C03628=1010.077,358.857,339.803,170.811,52.847,160.488
C03629=1010.084,359.105,339.765,170.821,52.843,160.489
C03630=1010.090,359.351,339.728,170.830,52.838,160.489
C03631=1010.098,359.598,339.690,170.839,52.835,160.490
C03632=1010.105,359.846,339.653,170.848,52.830,160.491
C03633=1010.112,360.093,339.616,170.857,52.827,160.492
C03634=1010.119,360.340,339.578,170.866,52.823,160.493
C03635=1010.126,360.587,339.541,170.876,52.819,160.494
C03636=1010.133,360.834,339.504,170.884,52.814,160.495
C03637=1010.140,361.081,339.466,170.893,52.811,160.495
C03638=1010.147,361.328,339.429,170.903,52.806,160.496
C03639=1010.155,361.575,339.391,170.912,52.803,160.497
C03640=1010.162,361.822,339.354,170.922,52.799,160.498
C03641=1010.169,362.069,339.316,170.930,52.795,160.499
C03642=1010.176,362.317,339.279,170.939,52.791,160.500
C03643=1010.184,362.564,339.241,170.949,52.787,160.501
C03644=1010.191,362.811,339.204,170.958,52.783,160.502
C03645=1010.198,363.058,339.166,170.968,52.779,160.503
C03646=1010.205,363.305,339.128,170.977,52.775,160.504
C03647=1010.213,363.552,339.090,170.987,52.771,160.505
C03648=1010.220,363.799,339.053,170.995,52.767,160.505
C03649=1010.227,364.046,339.015,171.005,52.763,160.506
C03650=1010.235,364.293,338.978,171.014,52.760,160.507
C03651=1010.242,364.539,338.939,171.023,52.756,160.508
C03652=1010.250,364.787,338.902,171.033,52.752,160.509
C03653=1010.257,365.034,338.864,171.042,52.749,160.510
C03654=1010.265,365.281,338.826,171.052,52.745,160.511
C03655=1010.272,365.528,338.788,171.061,52.741,160.512
C03656=1009.942,363.417,338.757,170.962,52.829,160.514
C03657=1009.935,363.169,338.794,170.952,52.833,160.513
C03658=1009.928,362.922,338.832,170.943,52.836,160.512
C03659=1009.920,362.675,338.869,170.934,52.840,160.511
C03660=1009.913,362.428,338.907,170.924,52.844,160.510
C03661=1009.906,362.181,338.944,170.915,52.848,160.509
C03662=1009.899,361.934,338.982,170.905,52.852,160.508
C03663=1009.891,361.687,339.019,170.897,52.856,160.508
C03664=1009.884,361.439,339.057,170.887,52.860,160.507
C03665=1009.877,361.192,339.094,170.878,52.864,160.506
C03666=1009.870,360.945,339.132,170.869,52.868,160.505
C03667=1009.863,360.698,339.169,170.859,52.872,160.504
C03668=1009.856,360.452,339.207,170.851,52.876,160.503
C03669=1009.849,360.205,339.244,170.842,52.880,160.502
C03670=1009.841,359.957,339.282,170.832,52.884,160.501
C03671=1009.834,359.710,339.318,170.823,52.888,160.501
C03672=1009.827,359.462,339.356,170.814,52.892,160.500
C03673=1009.821,359.216,339.393,170.805,52.896,160.499
C03674=1009.813,358.969,339.431,170.796,52.900,160.498
C03675=1009.806,358.721,339.468,170.786,52.904,160.497
C03676=1009.800,358.475,339.505,170.778,52.908,160.496
C03677=1009.793,358.227,339.541,170.769,52.913,160.496
C03678=1009.786,357.980,339.579,170.759,52.917,160.495
C03679=1009.779,357.733,339.615,170.751,52.921,160.494
C03680=1009.772,357.486,339.653,170.742,52.925,160.493
C03681=1009.765,357.238,339.690,170.733,52.929,160.492
C03682=1009.758,356.992,339.726,170.723,52.933,160.491
C03683=1009.751,356.744,339.763,170.715,52.937,160.491
C03684=1009.744,356.496,339.800,170.706,52.942,160.490
C03685=1009.737,356.250,339.837,170.697,52.946,160.489
C03686=1009.729,356.002,339.873,170.688,52.950,160.488
C03687=1009.723,355.755,339.910,170.679,52.954,160.487
C03688=1009.716,355.508,339.947,170.670,52.959,160.487
C03689=1009.710,355.284,339.979,170.662,52.962,160.486
C03690=1009.704,355.060,340.012,170.655,52.966,160.485
C03691=1009.697,354.837,340.046,170.646,52.970,160.485
C03692=1009.691,354.612,340.079,170.639,52.974,160.484
C03693=1009.684,354.389,340.112,170.630,52.978,160.483
C03694=1009.678,354.165,340.145,170.623,52.982,160.483
C03695=1009.673,353.941,340.178,170.615,52.986,160.482
C03696=1009.666,353.717,340.211,170.606,52.990,160.481
C03697=1009.660,353.470,340.247,170.598,52.994,160.481
C03698=1009.653,353.223,340.284,170.589,52.999,160.480
C03699=1009.646,352.976,340.320,170.581,53.003,160.479
C03700=1009.639,352.728,340.356,170.571,53.008,160.478
C03701=1009.633,352.480,340.392,170.563,53.012,160.478
C03702=1009.625,352.234,340.428,170.554,53.016,160.477
C03703=1009.619,351.986,340.465,170.546,53.020,160.476
C03704=1009.611,351.739,340.501,170.537,53.025,160.476
C03705=1009.605,351.492,340.536,170.528,53.030,160.475
C03706=1009.598,351.244,340.573,170.519,53.034,160.474
C03707=1009.591,350.997,340.609,170.511,53.038,160.474
C03708=1009.585,350.750,340.644,170.503,53.043,160.473
C03709=1009.578,350.503,340.681,170.494,53.047,160.472
C03710=1009.571,350.255,340.716,170.485,53.052,160.472
C03711=1009.565,350.008,340.753,170.477,53.057,160.471
C03712=1009.558,349.760,340.788,170.468,53.061,160.470
C03713=1009.552,349.513,340.824,170.459,53.065,160.470
C03714=1009.545,349.266,340.859,170.451,53.070,160.469
C03715=1009.538,349.019,340.896,170.443,53.074,160.468
C03716=1009.531,348.771,340.931,170.434,53.079,160.468
C03717=1009.525,348.524,340.968,170.425,53.084,160.467
C03718=1009.518,348.276,341.003,170.417,53.089,160.467
C03719=1009.512,348.029,341.039,170.409,53.093,160.466
C03720=1009.505,347.782,341.074,170.400,53.098,160.465
C03721=1009.499,347.534,341.110,170.392,53.102,160.465
C03722=1009.492,347.287,341.145,170.384,53.107,160.464
C03723=1009.486,347.039,341.181,170.374,53.111,160.463
C03724=1009.479,346.792,341.217,170.366,53.116,160.463
C03725=1009.472,346.545,341.252,170.358,53.121,160.462
C03726=1009.466,346.297,341.288,170.349,53.125,160.462
C03727=1009.459,346.050,341.323,170.341,53.130,160.461
C03728=1009.453,345.802,341.359,170.333,53.135,160.461
C03729=1009.447,345.555,341.394,170.325,53.139,160.460
C03730=1009.440,345.308,341.429,170.317,53.144,160.459
C03731=1009.434,345.060,341.465,170.309,53.149,160.459
C03732=1009.427,344.812,341.500,170.300,53.154,160.458
C03733=1009.420,344.565,341.535,170.291,53.159,160.457
C03734=1009.413,344.318,341.570,170.283,53.163,160.457
C03735=1009.408,344.071,341.605,170.275,53.168,160.456
C03736=1009.402,343.823,341.640,170.267,53.173,160.456
C03737=1009.395,343.575,341.675,170.259,53.178,160.455
C03738=1009.388,343.328,341.710,170.250,53.183,160.455
C03739=1009.381,343.081,341.745,170.242,53.187,160.454
C03740=1009.376,342.832,341.780,170.234,53.192,160.454
C03741=1009.369,342.586,341.815,170.226,53.197,160.453
C03742=1009.363,342.338,341.850,170.218,53.202,160.453
C03743=1009.356,342.090,341.885,170.209,53.207,160.452
C03744=1009.350,341.843,341.920,170.201,53.212,160.452
C03745=1009.344,341.596,341.955,170.193,53.216,160.451
C03746=1009.337,341.348,341.989,170.185,53.221,160.451
C03747=1009.331,341.101,342.025,170.177,53.226,160.450
C03748=1009.324,340.853,342.059,170.169,53.231,160.450
C03749=1009.318,340.606,342.094,170.161,53.236,160.449
C03750=1009.312,340.358,342.129,170.153,53.241,160.449
C03751=1009.306,340.110,342.164,170.145,53.246,160.448
C03752=1009.300,339.863,342.198,170.137,53.251,160.448
C03753=1009.291,339.530,342.244,170.125,53.259,160.447
C03754=1009.283,339.197,342.291,170.114,53.265,160.446
C03755=1009.275,338.864,342.338,170.104,53.271,160.446
C03756=1009.266,338.532,342.384,170.093,53.278,160.445
C03757=1009.260,338.285,342.419,170.085,53.284,160.445
C03758=1009.253,338.037,342.453,170.077,53.289,160.444
C03759=1009.247,337.790,342.487,170.069,53.293,160.444
C03760=1009.241,337.542,342.522,170.061,53.298,160.443
C03761=1009.235,337.295,342.556,170.053,53.304,160.443
C03762=1009.229,337.047,342.590,170.045,53.309,160.442
C03763=1009.223,336.799,342.624,170.037,53.314,160.442
C03764=1009.216,336.551,342.658,170.030,53.319,160.442
C03765=1009.211,336.304,342.693,170.021,53.324,160.441
C03766=1009.205,336.057,342.727,170.014,53.330,160.441
C03767=1009.198,335.809,342.761,170.006,53.335,160.440
C03768=1009.192,335.561,342.795,169.998,53.339,160.440
C03769=1009.185,335.314,342.829,169.990,53.345,160.440
C03770=1009.179,335.067,342.863,169.983,53.350,160.439
C03771=1009.173,334.819,342.897,169.975,53.355,160.439
C03772=1009.167,334.571,342.931,169.967,53.360,160.438
C03773=1009.161,334.323,342.965,169.960,53.366,160.438
C03774=1009.155,334.075,342.999,169.951,53.370,160.438
C03775=1009.149,333.828,343.033,169.944,53.376,160.437
C03776=1009.143,333.581,343.067,169.936,53.382,160.437
C03777=1009.138,333.333,343.101,169.928,53.386,160.436
C03778=1009.130,333.085,343.134,169.920,53.392,160.436
C03779=1009.125,332.838,343.168,169.912,53.397,160.436
C03780=1009.119,332.590,343.202,169.905,53.403,160.435
C03781=1009.113,332.343,343.236,169.897,53.408,160.435
C03782=1009.107,332.094,343.270,169.889,53.413,160.435
C03783=1009.101,331.847,343.304,169.881,53.419,160.434
C03784=1009.095,331.600,343.338,169.875,53.424,160.434
C03785=1009.090,331.352,343.371,169.867,53.429,160.434
C03786=1009.083,331.105,343.404,169.859,53.434,160.433
C03787=1009.077,330.856,343.438,169.851,53.440,160.433
C03788=1009.071,330.608,343.472,169.844,53.445,160.433
C03789=1009.065,330.361,343.505,169.836,53.450,160.432
C03790=1009.059,330.113,343.538,169.828,53.456,160.432
C03791=1009.054,329.865,343.572,169.820,53.461,160.432
C03792=1009.047,329.618,343.605,169.813,53.467,160.431
C03793=1009.042,329.371,343.638,169.805,53.473,160.431
C03794=1009.035,329.123,343.671,169.797,53.478,160.431
C03795=1009.030,328.875,343.705,169.791,53.483,160.430
C03796=1009.024,328.627,343.738,169.783,53.488,160.430
C03797=1009.018,328.380,343.771,169.775,53.494,160.430
C03798=1009.012,328.132,343.805,169.767,53.499,160.429
C03799=1009.006,327.884,343.838,169.760,53.505,160.429
C03800=1009.000,327.637,343.871,169.752,53.511,160.429
C03801=1008.995,327.389,343.904,169.744,53.516,160.428
C03802=1008.988,327.141,343.937,169.737,53.522,160.428
C03803=1008.983,326.893,343.970,169.730,53.527,160.428
C03804=1008.977,326.645,344.004,169.723,53.532,160.428
C03805=1008.971,326.398,344.036,169.715,53.538,160.427
C03806=1008.965,326.150,344.070,169.707,53.544,160.427
C03807=1008.960,325.902,344.103,169.700,53.549,160.427
C03808=1008.954,325.654,344.136,169.692,53.555,160.426
C03809=1008.948,325.407,344.169,169.686,53.561,160.427
C03810=1008.942,325.159,344.202,169.678,53.566,160.426
C03811=1008.937,324.912,344.235,169.671,53.572,160.426
C03812=1008.930,324.664,344.267,169.663,53.577,160.426
C03813=1008.923,324.327,344.311,169.653,53.585,160.425
C03814=1008.915,323.990,344.356,169.643,53.593,160.425
C03815=1008.906,323.652,344.399,169.633,53.600,160.425
C03816=1008.898,323.316,344.444,169.623,53.609,160.424
C03817=1008.892,323.067,344.476,169.615,53.614,160.424
C03818=1008.886,322.820,344.509,169.608,53.620,160.424
C03819=1008.881,322.572,344.541,169.601,53.626,160.424
C03820=1008.875,322.324,344.574,169.593,53.632,160.423
C03821=1008.869,322.076,344.606,169.585,53.637,160.423
C03822=1008.863,321.828,344.639,169.579,53.643,160.423
C03823=1008.857,321.581,344.670,169.572,53.649,160.423
C03824=1008.852,321.333,344.704,169.564,53.654,160.423
C03825=1008.846,321.085,344.736,169.557,53.661,160.422
C03826=1008.840,320.837,344.767,169.549,53.666,160.422
C03827=1008.834,320.590,344.800,169.542,53.672,160.422
C03828=1008.828,320.342,344.832,169.535,53.678,160.422
C03829=1008.823,320.094,344.864,169.528,53.683,160.422
C03830=1008.817,319.845,344.896,169.521,53.690,160.422
C03831=1008.811,319.598,344.929,169.513,53.695,160.421
C03832=1008.806,319.350,344.961,169.506,53.701,160.421
C03833=1008.800,319.102,344.993,169.498,53.707,160.421
C03834=1008.794,318.855,345.024,169.492,53.713,160.421
C03835=1008.788,318.606,345.056,169.484,53.719,160.420
C03836=1008.783,318.359,345.089,169.477,53.725,160.420
C03837=1008.777,318.111,345.121,169.470,53.731,160.420
C03838=1008.772,317.864,345.153,169.462,53.737,160.420
C03839=1008.766,317.615,345.185,169.456,53.743,160.420
C03840=1008.761,317.368,345.217,169.449,53.748,160.420
C03841=1008.755,317.120,345.249,169.441,53.755,160.420
C03842=1008.750,316.872,345.281,169.434,53.761,160.420
C03843=1008.744,316.624,345.313,169.428,53.766,160.419
C03844=1008.739,316.376,345.345,169.420,53.772,160.419
C03845=1008.733,316.128,345.377,169.413,53.778,160.419
C03846=1008.727,315.880,345.408,169.406,53.784,160.419
C03847=1008.723,315.632,345.441,169.398,53.790,160.419
C03848=1008.717,315.384,345.473,169.392,53.796,160.419
C03849=1008.711,315.137,345.504,169.385,53.802,160.419
C03850=1008.706,314.889,345.536,169.378,53.808,160.418
C03851=1008.700,314.641,345.568,169.370,53.815,160.418
C03852=1008.695,314.393,345.599,169.364,53.820,160.418
C03853=1008.690,314.145,345.631,169.357,53.826,160.418
C03854=1008.684,313.897,345.663,169.349,53.832,160.418
C03855=1008.679,313.649,345.695,169.342,53.839,160.418
C03856=1008.673,313.402,345.727,169.336,53.845,160.418
C03857=1008.668,313.154,345.758,169.328,53.850,160.418
C03858=1008.662,312.906,345.790,169.321,53.857,160.417
C03859=1008.658,312.658,345.822,169.315,53.862,160.417
C03860=1008.652,312.410,345.854,169.308,53.869,160.417
C03861=1008.647,312.162,345.884,169.301,53.875,160.417
C03862=1008.642,311.915,345.916,169.294,53.881,160.417
C03863=1008.636,311.666,345.948,169.288,53.887,160.417
C03864=1008.631,311.418,345.979,169.280,53.894,160.417
C03865=1008.626,311.170,346.011,169.273,53.899,160.417
C03866=1008.621,310.922,346.042,169.266,53.905,160.417
C03867=1008.616,310.675,346.074,169.259,53.911,160.417
C03868=1008.610,310.427,346.106,169.252,53.918,160.417
C03869=1008.605,310.179,346.137,169.245,53.924,160.417
C03870=1008.600,309.932,346.168,169.239,53.930,160.417
C03871=1008.594,309.683,346.200,169.232,53.936,160.416
C03872=1008.590,309.435,346.232,169.225,53.943,160.416
C03873=1008.583,309.104,346.273,169.216,53.951,160.417
C03874=1008.576,308.772,346.315,169.207,53.959,160.416
C03875=1008.569,308.441,346.357,169.197,53.967,160.416
C03876=1008.562,308.110,346.398,169.189,53.976,160.416
C03877=1008.557,307.861,346.429,169.182,53.982,160.416
C03878=1008.551,307.614,346.460,169.175,53.989,160.416
C03879=1008.546,307.365,346.491,169.168,53.994,160.416
C03880=1008.540,307.118,346.521,169.162,54.001,160.416
C03881=1008.535,306.870,346.552,169.155,54.008,160.416
C03882=1008.529,306.622,346.582,169.147,54.014,160.416
C03883=1008.524,306.374,346.613,169.141,54.020,160.416
C03884=1008.518,306.126,346.643,169.134,54.026,160.416
C03885=1008.513,305.878,346.674,169.127,54.033,160.416
C03886=1008.507,305.630,346.705,169.120,54.040,160.416
C03887=1008.502,305.382,346.736,169.114,54.046,160.416
C03888=1008.496,305.134,346.766,169.107,54.053,160.416
C03889=1008.492,304.885,346.796,169.100,54.059,160.416
C03890=1008.486,304.638,346.826,169.093,54.065,160.416
C03891=1008.481,304.390,346.857,169.087,54.071,160.416
C03892=1008.475,304.142,346.888,169.080,54.078,160.416
C03893=1008.470,303.894,346.919,169.073,54.085,160.416
C03894=1008.465,303.645,346.948,169.067,54.090,160.416
C03895=1008.460,303.397,346.979,169.060,54.098,160.416
C03896=1008.454,303.149,347.009,169.053,54.104,160.416
C03897=1008.450,302.901,347.039,169.047,54.111,160.416
C03898=1008.444,302.654,347.070,169.040,54.117,160.416
C03899=1008.439,302.405,347.101,169.033,54.123,160.416
C03900=1008.433,302.157,347.130,169.027,54.130,160.416
C03901=1008.428,301.909,347.161,169.020,54.136,160.416
C03902=1008.423,301.662,347.191,169.014,54.143,160.416
C03903=1008.418,301.413,347.221,169.007,54.149,160.416
C03904=1008.413,301.165,347.252,169.001,54.156,160.416
C03905=1008.408,300.916,347.282,168.994,54.162,160.416
C03906=1008.403,300.669,347.312,168.987,54.169,160.416
C03907=1008.398,300.421,347.342,168.981,54.175,160.416
C03908=1008.392,300.173,347.373,168.974,54.182,160.417
C03909=1008.386,299.863,347.410,168.966,54.190,160.416
C03910=1008.380,299.552,347.448,168.957,54.199,160.417
C03911=1008.373,299.242,347.486,168.949,54.207,160.417
C03912=1008.367,298.932,347.523,168.941,54.215,160.417
C03913=1008.125,299.698,347.065,168.938,54.244,160.423
C03914=1008.132,300.072,347.020,168.949,54.235,160.423
C03915=1008.141,300.446,346.974,168.958,54.225,160.423
C03916=1008.148,300.821,346.928,168.968,54.215,160.423
C03917=1008.156,301.195,346.883,168.978,54.206,160.423
C03918=1008.161,301.444,346.853,168.985,54.198,160.423
C03919=1008.166,301.692,346.822,168.991,54.193,160.423
C03920=1008.171,301.940,346.793,168.998,54.186,160.423
C03921=1008.176,302.188,346.762,169.005,54.179,160.423
C03922=1008.182,302.436,346.732,169.011,54.173,160.423
C03923=1008.187,302.685,346.701,169.018,54.166,160.422
C03924=1008.192,302.932,346.671,169.025,54.160,160.423
C03925=1008.197,303.180,346.641,169.031,54.154,160.423
C03926=1008.203,303.428,346.611,169.038,54.147,160.422
C03927=1008.208,303.676,346.580,169.045,54.141,160.423
C03928=1008.213,303.925,346.550,169.051,54.135,160.423
C03929=1008.218,304.172,346.520,169.058,54.128,160.423
C03930=1008.224,304.420,346.489,169.065,54.121,160.423
C03931=1008.229,304.668,346.458,169.072,54.115,160.423
C03932=1008.234,304.917,346.429,169.078,54.109,160.423
C03933=1008.239,305.165,346.398,169.085,54.103,160.423
C03934=1008.245,305.413,346.367,169.092,54.096,160.423
C03935=1008.250,305.661,346.336,169.098,54.090,160.423
C03936=1008.255,305.909,346.305,169.105,54.083,160.423
C03937=1008.261,306.157,346.276,169.112,54.077,160.423
C03938=1008.266,306.405,346.245,169.120,54.071,160.423
C03939=1008.271,306.652,346.215,169.125,54.064,160.423
C03940=1008.276,306.901,346.184,169.132,54.058,160.423
C03941=1008.282,307.148,346.154,169.139,54.051,160.423
C03942=1008.287,307.397,346.123,169.146,54.045,160.423
C03943=1008.293,307.644,346.092,169.153,54.039,160.423
C03944=1008.298,307.893,346.061,169.160,54.033,160.423
C03945=1008.304,308.141,346.031,169.167,54.026,160.423
C03946=1008.311,308.474,345.989,169.175,54.018,160.423
C03947=1008.318,308.807,345.947,169.185,54.010,160.423
C03948=1008.324,309.142,345.905,169.194,54.001,160.423
C03949=1008.331,309.475,345.863,169.203,53.993,160.423
C03950=1008.337,309.723,345.831,169.210,53.987,160.423
C03951=1008.342,309.971,345.800,169.217,53.980,160.424
C03952=1008.347,310.219,345.768,169.223,53.974,160.424
C03953=1008.352,310.467,345.737,169.230,53.968,160.424
C03954=1008.357,310.715,345.705,169.238,53.962,160.424
C03955=1008.362,310.963,345.674,169.245,53.956,160.424
C03956=1008.368,311.211,345.643,169.251,53.950,160.424
C03957=1008.372,311.459,345.611,169.259,53.944,160.424
C03958=1008.377,311.707,345.579,169.266,53.938,160.424
C03959=1008.383,311.954,345.548,169.272,53.932,160.424
C03960=1008.388,312.202,345.517,169.279,53.925,160.424
C03961=1008.394,312.450,345.485,169.287,53.920,160.425
C03962=1008.399,312.698,345.453,169.294,53.913,160.425
C03963=1008.404,312.946,345.422,169.300,53.908,160.425
C03964=1008.409,313.194,345.390,169.307,53.901,160.425
C03965=1008.414,313.441,345.358,169.314,53.895,160.425
C03966=1008.420,313.690,345.326,169.321,53.890,160.425
C03967=1008.426,313.938,345.295,169.328,53.883,160.425
C03968=1008.431,314.185,345.264,169.335,53.877,160.425
C03969=1008.436,314.433,345.232,169.342,53.871,160.425
C03970=1008.442,314.681,345.199,169.349,53.866,160.426
C03971=1008.447,314.929,345.168,169.356,53.859,160.426
C03972=1008.452,315.177,345.137,169.363,53.853,160.426
C03973=1008.458,315.425,345.105,169.371,53.847,160.426
C03974=1008.463,315.673,345.073,169.377,53.841,160.426
C03975=1008.469,315.920,345.041,169.384,53.835,160.426
C03976=1008.474,316.169,345.009,169.392,53.830,160.427
C03977=1008.479,316.416,344.977,169.399,53.823,160.427
C03978=1008.485,316.664,344.946,169.406,53.818,160.427
C03979=1008.491,316.912,344.913,169.413,53.812,160.427
C03980=1008.496,317.159,344.882,169.420,53.805,160.427
C03981=1008.501,317.408,344.849,169.428,53.800,160.427
C03982=1008.507,317.655,344.818,169.435,53.794,160.427
C03983=1008.513,317.904,344.786,169.441,53.788,160.428
C03984=1008.518,318.151,344.754,169.449,53.782,160.428
C03985=1008.524,318.399,344.722,169.456,53.776,160.428
C03986=1008.530,318.647,344.690,169.463,53.770,160.428
C03987=1008.535,318.895,344.658,169.470,53.765,160.428
C03988=1008.540,319.143,344.626,169.477,53.759,160.428
C03989=1008.546,319.391,344.593,169.485,53.753,160.429
C03990=1008.552,319.638,344.561,169.492,53.747,160.429
C03991=1008.558,319.886,344.529,169.500,53.741,160.429
C03992=1008.563,320.134,344.498,169.507,53.735,160.429
C03993=1008.568,320.382,344.465,169.513,53.730,160.429
C03994=1008.575,320.630,344.432,169.521,53.724,160.430
C03995=1008.580,320.877,344.401,169.528,53.718,160.430
C03996=1008.586,321.126,344.369,169.536,53.712,160.430
C03997=1008.592,321.374,344.337,169.543,53.706,160.430
C03998=1008.598,321.621,344.304,169.550,53.701,160.430
C03999=1008.603,321.869,344.272,169.557,53.695,160.431
C04000=1008.609,322.117,344.239,169.565,53.689,160.431
C04001=1008.615,322.364,344.207,169.572,53.683,160.431
C04002=1008.621,322.613,344.175,169.580,53.677,160.431
C04003=1008.627,322.860,344.143,169.587,53.672,160.432
C04004=1008.632,323.109,344.110,169.595,53.666,160.432
C04005=1008.638,323.356,344.078,169.601,53.660,160.432
C04006=1008.647,323.695,344.034,169.612,53.653,160.433
C04007=1008.654,324.035,343.989,169.623,53.645,160.433
C04008=1008.662,324.374,343.944,169.632,53.637,160.433
C04009=1008.671,324.713,343.900,169.642,53.629,160.434
C04010=1008.677,324.961,343.867,169.650,53.624,160.434
C04011=1008.682,325.209,343.835,169.658,53.618,160.434
C04012=1008.687,325.457,343.802,169.665,53.613,160.434
C04013=1008.693,325.704,343.769,169.671,53.607,160.434
C04014=1008.699,325.952,343.736,169.679,53.601,160.435
C04015=1008.705,326.200,343.702,169.687,53.596,160.435
C04016=1008.711,326.448,343.670,169.694,53.590,160.435
C04017=1008.716,326.695,343.636,169.702,53.584,160.436
C04018=1008.723,326.943,343.604,169.710,53.579,160.436
C04019=1008.728,327.191,343.570,169.716,53.574,160.436
C04020=1008.734,327.439,343.537,169.724,53.569,160.437
C04021=1008.740,327.686,343.504,169.732,53.563,160.437
C04022=1008.745,327.934,343.471,169.740,53.558,160.437
C04023=1008.751,328.182,343.438,169.747,53.552,160.438
C04024=1008.757,328.429,343.405,169.755,53.546,160.438
C04025=1008.762,328.677,343.372,169.763,53.541,160.438
C04026=1008.769,328.924,343.338,169.770,53.535,160.438
C04027=1008.775,329.173,343.305,169.777,53.530,160.439
C04028=1008.781,329.421,343.271,169.784,53.524,160.439
C04029=1008.787,329.668,343.239,169.793,53.520,160.440
C04030=1008.793,329.916,343.205,169.800,53.514,160.440
C04031=1008.798,330.163,343.171,169.808,53.508,160.440
C04032=1008.805,330.411,343.138,169.815,53.503,160.440
C04033=1008.810,330.659,343.105,169.823,53.497,160.441
C04034=1008.816,330.906,343.071,169.831,53.492,160.441
C04035=1008.822,331.154,343.038,169.839,53.487,160.442
C04036=1008.828,331.402,343.005,169.846,53.481,160.442
C04037=1008.834,331.650,342.971,169.855,53.476,160.442
C04038=1008.840,331.898,342.937,169.861,53.471,160.443
C04039=1008.846,332.145,342.903,169.869,53.465,160.443
C04040=1008.851,332.393,342.870,169.877,53.461,160.443
C04041=1008.858,332.640,342.836,169.885,53.455,160.444
C04042=1008.864,332.887,342.802,169.893,53.450,160.444
C04043=1008.870,333.136,342.769,169.900,53.444,160.444
C04044=1008.876,333.383,342.735,169.908,53.439,160.445
C04045=1008.882,333.630,342.700,169.916,53.434,160.445
C04046=1008.887,333.878,342.667,169.924,53.428,160.446
C04047=1008.894,334.126,342.633,169.932,53.423,160.446
C04048=1008.900,334.373,342.599,169.939,53.418,160.446
C04049=1008.905,334.621,342.565,169.948,53.413,160.447
C04050=1008.912,334.869,342.532,169.955,53.407,160.447
C04051=1008.918,335.116,342.497,169.963,53.403,160.448
C04052=1008.924,335.363,342.463,169.971,53.397,160.448
C04053=1008.931,335.611,342.429,169.979,53.392,160.449
C04054=1008.936,335.859,342.395,169.986,53.388,160.449
C04055=1008.943,336.107,342.361,169.994,53.382,160.449
C04056=1008.948,336.355,342.327,170.002,53.377,160.450
C04057=1008.954,336.602,342.293,170.009,53.371,160.450
C04058=1008.961,336.850,342.259,170.018,53.367,160.451
C04059=1008.967,337.097,342.225,170.026,53.362,160.451
C04060=1008.974,337.345,342.191,170.033,53.356,160.451
C04061=1008.980,337.592,342.157,170.041,53.351,160.452
C04062=1008.986,337.840,342.122,170.049,53.346,160.452
C04063=1008.992,338.087,342.088,170.058,53.341,160.453
C04064=1008.998,338.335,342.053,170.066,53.337,160.453
C04065=1009.004,338.582,342.019,170.073,53.331,160.454
C04066=1009.013,338.917,341.972,170.084,53.324,160.454
C04067=1009.021,339.252,341.925,170.096,53.317,160.455
C04068=1009.029,339.588,341.879,170.107,53.311,160.456
C04069=1009.038,339.922,341.832,170.117,53.304,160.457
C04070=1009.044,340.169,341.797,170.125,53.299,160.457
C04071=1009.050,340.418,341.762,170.134,53.294,160.458
C04072=1009.056,340.664,341.727,170.141,53.289,160.458
C04073=1009.063,340.912,341.693,170.149,53.284,160.458
C04074=1009.069,341.160,341.658,170.157,53.279,160.459
C04075=1009.075,341.407,341.624,170.165,53.274,160.459
C04076=1009.082,341.654,341.589,170.174,53.269,160.460
C04077=1009.088,341.903,341.554,170.182,53.264,160.460
C04078=1009.094,342.149,341.519,170.190,53.259,160.461
C04079=1009.100,342.397,341.484,170.198,53.255,160.462
C04080=1009.107,342.645,341.449,170.206,53.250,160.462
C04081=1009.113,342.892,341.413,170.216,53.245,160.463
C04082=1009.120,343.140,341.379,170.224,53.240,160.463
C04083=1009.126,343.387,341.344,170.232,53.235,160.464
C04084=1009.133,343.634,341.309,170.240,53.230,160.464
C04085=1009.139,343.882,341.275,170.248,53.226,160.465
C04086=1009.145,344.130,341.239,170.256,53.221,160.466
C04087=1009.152,344.377,341.204,170.265,53.216,160.466
C04088=1009.159,344.625,341.169,170.273,53.211,160.467
C04089=1009.165,344.871,341.134,170.281,53.207,160.467
C04090=1009.171,345.119,341.098,170.289,53.202,160.468
C04091=1009.177,345.367,341.064,170.297,53.197,160.468
C04092=1009.184,345.614,341.029,170.307,53.192,160.469
C04093=1009.190,345.862,340.993,170.315,53.187,160.469
C04094=1009.197,346.109,340.957,170.323,53.183,160.470
C04095=1009.204,346.356,340.922,170.331,53.178,160.471
C04096=1009.210,346.604,340.886,170.339,53.173,160.471
C04097=1009.217,346.851,340.851,170.348,53.169,160.472
C04098=1009.223,347.099,340.815,170.356,53.164,160.472
C04099=1009.230,347.346,340.780,170.365,53.160,160.473
C04100=1009.236,347.594,340.744,170.373,53.155,160.474
C04101=1009.243,347.841,340.709,170.382,53.150,160.475
C04102=1009.249,348.088,340.673,170.390,53.146,160.475
C04103=1009.255,348.336,340.638,170.399,53.141,160.476
C04104=1009.262,348.583,340.601,170.407,53.136,160.476
C04105=1009.269,348.830,340.566,170.415,53.132,160.477
C04106=1009.275,349.078,340.530,170.424,53.127,160.477
C04107=1009.282,349.325,340.495,170.432,53.123,160.478
C04108=1009.288,349.573,340.459,170.442,53.119,160.479
C04109=1009.295,349.820,340.423,170.450,53.114,160.480
C04110=1009.302,350.067,340.388,170.458,53.109,160.480
C04111=1009.308,350.314,340.351,170.467,53.105,160.481
C04112=1009.315,350.562,340.316,170.475,53.100,160.481
C04113=1009.322,350.809,340.279,170.485,53.096,160.482
C04114=1009.329,351.057,340.244,170.493,53.091,160.483
C04115=1009.335,351.304,340.208,170.501,53.087,160.484
C04116=1009.342,351.551,340.172,170.510,53.082,160.484
C04117=1009.349,351.799,340.136,170.518,53.078,160.485
C04118=1009.356,352.046,340.100,170.528,53.074,160.486
C04119=1009.362,352.293,340.064,170.536,53.069,160.487
C04120=1009.369,352.540,340.028,170.544,53.064,160.487
C04121=1009.376,352.788,339.991,170.553,53.060,160.488
C04122=1009.382,353.035,339.955,170.563,53.056,160.489
C04123=1009.389,353.282,339.918,170.571,53.051,160.489
C04124=1009.396,353.529,339.882,170.580,53.047,160.490
C04125=1009.403,353.776,339.846,170.588,53.043,160.491
C04126=1009.414,354.175,339.788,170.602,53.036,160.492
C04127=1009.425,354.573,339.728,170.617,53.029,160.493
C04128=1009.436,354.971,339.671,170.631,53.022,160.494
C04129=1009.447,355.369,339.612,170.645,53.015,160.496
C04130=1009.454,355.616,339.575,170.654,53.011,160.496
C04131=1009.461,355.864,339.538,170.664,53.006,160.497
C04132=1009.468,356.110,339.502,170.672,53.002,160.498
C04133=1009.475,356.357,339.465,170.681,52.998,160.499
C04134=1009.481,356.604,339.429,170.691,52.994,160.500
C04135=1009.488,356.852,339.392,170.699,52.990,160.500
C04136=1009.496,357.098,339.355,170.708,52.986,160.501
C04137=1009.503,357.346,339.318,170.717,52.981,160.502
C04138=1009.510,357.594,339.282,170.726,52.977,160.503
C04139=1009.516,357.840,339.244,170.735,52.973,160.504
C04140=1009.523,358.088,339.208,170.744,52.968,160.505
C04141=1009.530,358.335,339.170,170.753,52.964,160.505
C04142=1009.537,358.582,339.134,170.762,52.961,160.506
C04143=1009.544,358.829,339.096,170.771,52.956,160.507
C04144=1009.551,359.077,339.059,170.780,52.953,160.508
C04145=1009.558,359.324,339.022,170.789,52.948,160.509
C04146=1009.565,359.571,338.985,170.799,52.944,160.510
C04147=1009.572,359.818,338.947,170.807,52.940,160.510
C04148=1009.579,360.064,338.910,170.817,52.937,160.511
C04149=1009.586,360.312,338.873,170.826,52.932,160.512
C04150=1009.593,360.559,338.836,170.835,52.928,160.513
C04151=1009.600,360.806,338.798,170.845,52.924,160.514
C04152=1009.607,361.053,338.761,170.854,52.920,160.515
C04153=1009.614,361.300,338.723,170.862,52.916,160.516
C04154=1009.289,359.188,338.687,170.765,53.003,160.517
C04155=1009.283,358.942,338.724,170.756,53.007,160.517
C04156=1009.275,358.695,338.762,170.746,53.011,160.516
C04157=1009.269,358.447,338.799,170.738,53.016,160.515
C04158=1009.262,358.201,338.836,170.729,53.019,160.514
C04159=1009.255,357.953,338.873,170.719,53.024,160.513
C04160=1009.248,357.707,338.909,170.711,53.028,160.512
C04161=1009.241,357.459,338.946,170.702,53.032,160.511
C04162=1009.234,357.211,338.983,170.692,53.036,160.511
C04163=1009.227,356.964,339.019,170.684,53.040,160.510
C04164=1009.219,356.717,339.056,170.675,53.045,160.509
C04165=1009.213,356.470,339.093,170.665,53.049,160.508
C04166=1009.206,356.223,339.129,170.656,53.053,160.507
C04167=1009.200,355.976,339.166,170.648,53.057,160.507
C04168=1009.192,355.728,339.202,170.638,53.062,160.506
C04169=1009.185,355.482,339.239,170.630,53.066,160.505
C04170=1009.179,355.234,339.276,170.621,53.070,160.504
C04171=1009.169,354.885,339.326,170.609,53.076,160.503
C04172=1009.159,354.536,339.378,170.595,53.082,160.502
C04173=1009.149,354.185,339.430,170.583,53.089,160.501
C04174=1009.140,353.837,339.481,170.571,53.095,160.500
C04175=1009.133,353.588,339.518,170.562,53.099,160.499
C04176=1009.126,353.341,339.553,170.553,53.103,160.498
C04177=1009.120,353.094,339.590,170.544,53.108,160.498
C04178=1009.113,352.847,339.627,170.535,53.112,160.497
C04179=1009.106,352.600,339.663,170.527,53.116,160.496
C04180=1009.100,352.353,339.699,170.518,53.120,160.495
C04181=1009.094,352.105,339.735,170.510,53.125,160.495
C04182=1009.086,351.858,339.771,170.501,53.130,160.494
C04183=1009.079,351.611,339.807,170.492,53.134,160.493
C04184=1009.073,351.363,339.842,170.484,53.138,160.493
C04185=1009.066,351.117,339.878,170.475,53.143,160.492
C04186=1009.059,350.868,339.914,170.466,53.148,160.491
C04187=1009.052,350.621,339.950,170.457,53.152,160.491
C04188=1009.046,350.374,339.986,170.449,53.156,160.490
C04189=1009.039,350.127,340.022,170.440,53.161,160.489
C04190=1009.033,349.879,340.058,170.432,53.165,160.489
C04191=1009.026,349.632,340.093,170.423,53.170,160.488
C04192=1009.019,349.384,340.130,170.414,53.174,160.487
C04193=1009.012,349.137,340.165,170.406,53.179,160.487
C04194=1009.006,348.890,340.201,170.397,53.183,160.486
C04195=1008.999,348.642,340.236,170.389,53.188,160.485
C04196=1008.993,348.395,340.272,170.381,53.193,160.485
C04197=1008.987,348.147,340.307,170.372,53.198,160.484
C04198=1008.980,347.900,340.344,170.363,53.202,160.483
C04199=1008.973,347.653,340.379,170.355,53.207,160.483
C04200=1008.967,347.405,340.414,170.346,53.211,160.482
C04201=1008.961,347.158,340.450,170.338,53.216,160.481
C04202=1008.955,346.910,340.485,170.330,53.220,160.481
C04203=1008.948,346.663,340.520,170.322,53.225,160.480
C04204=1008.941,346.416,340.557,170.312,53.230,160.479
C04205=1008.935,346.168,340.592,170.304,53.235,160.479
C04206=1008.928,345.921,340.627,170.296,53.239,160.478
C04207=1008.922,345.673,340.663,170.287,53.244,160.478
C04208=1008.916,345.427,340.698,170.279,53.249,160.477
C04209=1008.909,345.179,340.732,170.271,53.253,160.476
C04210=1008.903,344.931,340.768,170.263,53.258,160.476
C04211=1008.896,344.684,340.803,170.255,53.263,160.475
C04212=1008.890,344.436,340.838,170.246,53.268,160.475
C04213=1008.883,344.189,340.873,170.237,53.272,160.474
C04214=1008.877,343.941,340.908,170.229,53.277,160.473
C04215=1008.871,343.694,340.943,170.221,53.282,160.473
C04216=1008.864,343.447,340.978,170.213,53.287,160.472
C04217=1008.858,343.199,341.013,170.205,53.292,160.472
C04218=1008.851,342.951,341.048,170.196,53.296,160.471
C04219=1008.846,342.704,341.083,170.188,53.301,160.471
C04220=1008.839,342.456,341.117,170.180,53.306,160.470
C04221=1008.832,342.209,341.153,170.172,53.311,160.470
C04222=1008.826,341.961,341.187,170.164,53.316,160.469
C04223=1008.821,341.714,341.222,170.156,53.321,160.469
C04224=1008.814,341.466,341.257,170.147,53.326,160.468
C04225=1008.808,341.219,341.292,170.139,53.330,160.468
C04226=1008.801,340.971,341.326,170.131,53.335,160.467
C04227=1008.795,340.724,341.361,170.123,53.340,160.467
C04228=1008.789,340.477,341.395,170.115,53.345,160.466
C04229=1008.783,340.229,341.431,170.107,53.350,160.466
C04230=1008.776,339.981,341.465,170.099,53.355,160.465
C04231=1008.768,339.644,341.512,170.087,53.362,160.464
C04232=1008.760,339.307,341.559,170.077,53.369,160.464
C04233=1008.751,338.969,341.607,170.066,53.376,160.463
C04234=1008.743,338.632,341.653,170.054,53.382,160.462
C04235=1008.737,338.385,341.687,170.046,53.388,160.462
C04236=1008.730,338.137,341.722,170.038,53.393,160.461
C04237=1008.725,337.890,341.756,170.030,53.398,160.461
C04238=1008.718,337.642,341.791,170.023,53.402,160.460
C04239=1008.712,337.395,341.825,170.015,53.407,160.460
C04240=1008.706,337.147,341.859,170.007,53.413,160.460
C04241=1008.700,336.900,341.893,169.999,53.417,160.459
C04242=1008.694,336.652,341.927,169.991,53.422,160.458
C04243=1008.688,336.404,341.962,169.983,53.428,160.458
C04244=1008.682,336.156,341.995,169.975,53.433,160.458
C04245=1008.676,335.908,342.029,169.967,53.438,160.457
C04246=1008.669,335.661,342.063,169.959,53.443,160.457
C04247=1008.663,335.414,342.097,169.951,53.448,160.456
C04248=1008.657,335.166,342.131,169.944,53.454,160.456
C04249=1008.651,334.918,342.165,169.936,53.459,160.455
C04250=1008.645,334.671,342.199,169.928,53.464,160.455
C04251=1008.639,334.423,342.233,169.920,53.469,160.455
C04252=1008.633,334.176,342.267,169.912,53.474,160.454
C04253=1008.627,333.928,342.301,169.904,53.480,160.454
C04254=1008.621,333.680,342.335,169.896,53.485,160.453
C04255=1008.614,333.433,342.368,169.888,53.490,160.453
C04256=1008.609,333.185,342.402,169.880,53.495,160.452
C04257=1008.603,332.938,342.436,169.873,53.501,160.452
C04258=1008.597,332.690,342.469,169.865,53.506,160.452
C04259=1008.591,332.442,342.503,169.857,53.511,160.451
C04260=1008.586,332.195,342.537,169.849,53.517,160.451
C04261=1008.579,331.947,342.571,169.842,53.521,160.451
C04262=1008.574,331.699,342.604,169.835,53.527,160.450
C04263=1008.568,331.451,342.638,169.826,53.532,160.450
C04264=1008.562,331.204,342.671,169.819,53.537,160.449
C04265=1008.556,330.956,342.705,169.811,53.543,160.449
C04266=1008.550,330.709,342.739,169.803,53.548,160.449
C04267=1008.544,330.461,342.771,169.795,53.554,160.448
C04268=1008.538,330.213,342.805,169.788,53.559,160.448
C04269=1008.533,329.966,342.839,169.780,53.565,160.448
C04270=1008.526,329.718,342.871,169.772,53.570,160.447
C04271=1008.521,329.470,342.905,169.765,53.575,160.447
C04272=1008.515,329.222,342.938,169.758,53.580,160.447
C04273=1008.509,328.975,342.971,169.750,53.586,160.446
C04274=1008.503,328.727,343.004,169.743,53.592,160.446
C04275=1008.497,328.479,343.037,169.734,53.597,160.446
C04276=1008.491,328.231,343.070,169.727,53.602,160.445
C04277=1008.486,327.984,343.104,169.719,53.608,160.445
C04278=1008.479,327.737,343.137,169.712,53.613,160.445
C04279=1008.474,327.489,343.170,169.704,53.619,160.444
C04280=1008.468,327.241,343.204,169.697,53.624,160.444
C04281=1008.462,326.992,343.236,169.690,53.630,160.444
C04282=1008.457,326.745,343.269,169.682,53.635,160.443
C04283=1008.450,326.497,343.302,169.674,53.641,160.443
C04284=1008.445,326.249,343.335,169.667,53.647,160.443
C04285=1008.440,326.002,343.368,169.659,53.652,160.443
C04286=1008.434,325.754,343.401,169.653,53.657,160.442
C04287=1008.428,325.506,343.434,169.645,53.663,160.442
C04288=1008.422,325.258,343.468,169.637,53.669,160.442
C04289=1008.416,325.010,343.500,169.630,53.674,160.441
C04290=1008.412,324.763,343.533,169.622,53.680,160.441
C04291=1008.403,324.421,343.577,169.612,53.687,160.441
C04292=1008.395,324.080,343.622,169.602,53.695,160.440
C04293=1008.387,323.738,343.666,169.592,53.703,160.440
C04294=1008.379,323.396,343.711,169.581,53.711,160.440
C04295=1008.373,323.148,343.744,169.573,53.716,160.439
C04296=1008.367,322.900,343.776,169.566,53.722,160.439
C04297=1008.361,322.653,343.808,169.559,53.728,160.439
C04298=1008.355,322.405,343.840,169.552,53.734,160.439
C04299=1008.349,322.157,343.872,169.544,53.739,160.438
C04300=1008.344,321.910,343.905,169.536,53.745,160.438
C04301=1008.338,321.661,343.937,169.529,53.751,160.438
C04302=1008.332,321.413,343.969,169.523,53.756,160.438
C04303=1008.327,321.166,344.002,169.515,53.762,160.437
C04304=1008.321,320.918,344.034,169.508,53.768,160.437
C04305=1008.315,320.670,344.066,169.500,53.774,160.437
C04306=1008.310,320.422,344.098,169.493,53.779,160.437
C04307=1008.304,320.174,344.130,169.486,53.785,160.437
C04308=1008.298,319.927,344.163,169.479,53.791,160.436
C04309=1008.292,319.679,344.195,169.471,53.797,160.436
C04310=1008.287,319.431,344.226,169.464,53.803,160.436
C04311=1008.282,319.183,344.259,169.456,53.808,160.436
C04312=1008.276,318.935,344.291,169.450,53.814,160.436
C04313=1008.270,318.687,344.323,169.443,53.820,160.435
C04314=1008.265,318.439,344.354,169.435,53.826,160.435
C04315=1008.259,318.191,344.386,169.428,53.832,160.435
C04316=1008.253,317.944,344.418,169.420,53.838,160.435
C04317=1008.248,317.695,344.451,169.414,53.843,160.435
C04318=1008.243,317.448,344.482,169.406,53.849,160.434
C04319=1008.237,317.200,344.514,169.399,53.855,160.434
C04320=1008.231,316.952,344.546,169.392,53.861,160.434
C04321=1008.226,316.704,344.578,169.385,53.867,160.434
C04322=1008.220,316.456,344.610,169.378,53.872,160.434
C04323=1008.215,316.208,344.642,169.371,53.879,160.433
C04324=1008.210,315.961,344.673,169.363,53.885,160.433
C04325=1008.204,315.713,344.706,169.357,53.890,160.433
C04326=1008.199,315.465,344.737,169.350,53.897,160.433
C04327=1008.194,315.217,344.768,169.342,53.902,160.433
C04328=1008.188,314.970,344.800,169.335,53.909,160.433
C04329=1008.183,314.721,344.832,169.329,53.915,160.433
C04330=1008.178,314.474,344.864,169.321,53.920,160.432
C04331=1008.173,314.225,344.895,169.314,53.926,160.432
C04332=1008.167,313.978,344.927,169.307,53.933,160.432
C04333=1008.161,313.730,344.959,169.300,53.938,160.432
C04334=1008.156,313.482,344.990,169.293,53.944,160.432
C04335=1008.151,313.234,345.022,169.286,53.951,160.432
C04336=1008.146,312.986,345.054,169.279,53.956,160.431
C04337=1008.141,312.739,345.085,169.272,53.962,160.431
C04338=1008.135,312.490,345.117,169.265,53.969,160.431
C04339=1008.130,312.242,345.148,169.258,53.975,160.431
C04340=1008.125,311.994,345.179,169.251,53.980,160.431
C04341=1008.120,311.746,345.211,169.244,53.986,160.431
C04342=1008.115,311.498,345.242,169.237,53.993,160.431
C04343=1008.109,311.251,345.274,169.231,53.999,160.431
C04344=1008.104,311.003,345.305,169.224,54.005,160.431
C04345=1008.099,310.755,345.337,169.216,54.011,160.431
C04346=1008.094,310.507,345.368,169.210,54.017,160.430
C04347=1008.089,310.259,345.400,169.203,54.023,160.430
C04348=1008.084,310.011,345.431,169.195,54.029,160.430
C04349=1008.079,309.764,345.462,169.189,54.035,160.430
C04350=1008.074,309.515,345.493,169.182,54.041,160.430
C04351=1008.066,309.180,345.536,169.172,54.050,160.430
C04352=1008.060,308.843,345.578,169.163,54.058,160.430
C04353=1008.053,308.508,345.621,169.155,54.066,160.430
C04354=1008.046,308.172,345.663,169.145,54.075,160.429
C04355=1008.040,307.924,345.694,169.138,54.081,160.429
C04356=1008.036,307.675,345.724,169.131,54.087,160.429
C04357=1008.030,307.427,345.754,169.124,54.093,160.429
C04358=1008.025,307.179,345.785,169.117,54.100,160.429
C04359=1008.019,306.932,345.816,169.110,54.106,160.429
C04360=1008.014,306.683,345.846,169.104,54.112,160.429
C04361=1008.008,306.436,345.877,169.097,54.119,160.429
C04362=1008.003,306.187,345.908,169.090,54.125,160.429
C04363=1007.997,305.939,345.937,169.083,54.132,160.429
C04364=1007.992,305.691,345.968,169.077,54.137,160.429
C04365=1007.987,305.444,345.998,169.070,54.144,160.429
C04366=1007.982,305.196,346.029,169.063,54.150,160.429
C04367=1007.977,304.947,346.060,169.056,54.156,160.429
C04368=1007.971,304.699,346.090,169.050,54.163,160.429
C04369=1007.966,304.451,346.121,169.043,54.169,160.429
C04370=1007.961,304.203,346.151,169.036,54.175,160.429
C04371=1007.956,303.955,346.181,169.029,54.182,160.429
C04372=1007.951,303.707,346.211,169.023,54.189,160.429
C04373=1007.945,303.459,346.242,169.017,54.195,160.429
C04374=1007.940,303.211,346.272,169.009,54.201,160.429
C04375=1007.935,302.963,346.303,169.002,54.207,160.429
C04376=1007.930,302.715,346.332,168.997,54.214,160.429
C04377=1007.925,302.467,346.363,168.989,54.220,160.429
C04378=1007.919,302.218,346.393,168.982,54.227,160.429
C04379=1007.915,301.996,346.420,168.976,54.233,160.429
C04380=1007.911,301.772,346.448,168.971,54.238,160.429
C04381=1007.906,301.549,346.475,168.965,54.244,160.429
C04382=1007.901,301.326,346.502,168.959,54.250,160.429
C04383=1007.897,301.103,346.528,168.953,54.256,160.429
C04384=1007.892,300.880,346.556,168.947,54.261,160.429
C04385=1007.888,300.657,346.583,168.941,54.267,160.429
C04386=1007.883,300.433,346.610,168.935,54.273,160.429
C04387=1007.641,301.143,346.158,168.932,54.301,160.434
C04388=1007.646,301.419,346.125,168.939,54.293,160.434
C04389=1007.652,301.696,346.091,168.946,54.286,160.434
C04390=1007.657,301.973,346.058,168.954,54.279,160.434
C04391=1007.663,302.250,346.024,168.961,54.272,160.434
C04392=1007.668,302.497,345.994,168.968,54.266,160.434
C04393=1007.673,302.746,345.964,168.975,54.259,160.434
C04394=1007.679,302.993,345.933,168.981,54.253,160.434
C04395=1007.684,303.242,345.903,168.988,54.247,160.434
C04396=1007.689,303.489,345.873,168.995,54.240,160.434
C04397=1007.694,303.737,345.842,169.001,54.234,160.434
C04398=1007.699,303.986,345.813,169.008,54.227,160.434
C04399=1007.704,304.234,345.782,169.015,54.221,160.434
C04400=1007.710,304.481,345.752,169.021,54.215,160.434
C04401=1007.714,304.730,345.721,169.028,54.209,160.435
C04402=1007.720,304.978,345.691,169.035,54.202,160.435
C04403=1007.725,305.227,345.661,169.041,54.196,160.435
C04404=1007.731,305.474,345.631,169.049,54.190,160.435
C04405=1007.735,305.722,345.600,169.056,54.184,160.435
C04406=1007.741,305.970,345.570,169.062,54.178,160.435
C04407=1007.746,306.218,345.539,169.069,54.171,160.435
C04408=1007.752,306.466,345.509,169.076,54.164,160.435
C04409=1007.757,306.714,345.478,169.082,54.158,160.435
C04410=1007.762,306.962,345.448,169.089,54.152,160.435
C04411=1007.768,307.210,345.417,169.096,54.146,160.435
C04412=1007.772,307.459,345.387,169.102,54.140,160.435
C04413=1007.778,307.707,345.356,169.109,54.133,160.435
C04414=1007.783,307.955,345.325,169.117,54.127,160.435
C04415=1007.789,308.203,345.295,169.124,54.121,160.435
C04416=1007.796,308.541,345.253,169.132,54.113,160.436
C04417=1007.802,308.878,345.210,169.142,54.105,160.436
C04418=1007.810,309.217,345.167,169.152,54.096,160.436
C04419=1007.816,309.555,345.125,169.161,54.087,160.436
C04420=1007.821,309.803,345.093,169.168,54.082,160.436
C04421=1007.826,310.051,345.062,169.175,54.076,160.436
C04422=1007.831,310.299,345.030,169.182,54.070,160.437
C04423=1007.836,310.547,344.999,169.188,54.064,160.436
C04424=1007.841,310.795,344.969,169.195,54.057,160.437
C04425=1007.847,311.042,344.937,169.203,54.052,160.437
C04426=1007.851,311.291,344.905,169.209,54.046,160.437
C04427=1007.856,311.538,344.874,169.216,54.039,160.437
C04428=1007.861,311.787,344.843,169.223,54.033,160.437
C04429=1007.867,312.034,344.811,169.230,54.028,160.437
C04430=1007.873,312.283,344.780,169.237,54.021,160.437
C04431=1007.878,312.530,344.748,169.244,54.015,160.438
C04432=1007.883,312.778,344.716,169.250,54.009,160.438
C04433=1007.888,313.026,344.685,169.258,54.004,160.438
C04434=1007.893,313.274,344.653,169.265,53.997,160.438
C04435=1007.898,313.522,344.622,169.273,53.992,160.438
C04436=1007.904,313.770,344.591,169.279,53.986,160.438
C04437=1007.909,314.017,344.559,169.286,53.979,160.438
C04438=1007.914,314.266,344.527,169.294,53.974,160.439
C04439=1007.919,314.514,344.495,169.300,53.968,160.439
C04440=1007.925,314.761,344.464,169.307,53.961,160.439
C04441=1007.930,315.009,344.432,169.315,53.956,160.439
C04442=1007.936,315.258,344.401,169.322,53.949,160.439
C04443=1007.941,315.505,344.369,169.328,53.944,160.440
C04444=1007.946,315.753,344.337,169.336,53.938,160.440
C04445=1007.951,316.000,344.305,169.343,53.932,160.440
C04446=1007.957,316.249,344.273,169.349,53.926,160.440
C04447=1007.962,316.497,344.242,169.357,53.921,160.440
C04448=1007.968,316.744,344.211,169.364,53.914,160.440
C04449=1007.974,316.992,344.179,169.372,53.909,160.441
C04450=1007.978,317.240,344.146,169.378,53.903,160.441
C04451=1007.984,317.489,344.114,169.386,53.897,160.441
C04452=1007.990,317.736,344.083,169.393,53.891,160.441
C04453=1007.995,317.984,344.051,169.400,53.885,160.441
C04454=1008.001,318.232,344.019,169.407,53.879,160.441
C04455=1008.006,318.480,343.987,169.414,53.874,160.442
C04456=1008.012,318.728,343.955,169.422,53.868,160.442
C04457=1008.017,318.975,343.923,169.429,53.862,160.442
C04458=1008.022,319.223,343.891,169.437,53.856,160.443
C04459=1008.028,319.471,343.859,169.443,53.851,160.443
C04460=1008.034,319.719,343.828,169.450,53.845,160.443
C04461=1008.039,319.967,343.795,169.458,53.839,160.443
C04462=1008.045,320.215,343.763,169.466,53.833,160.444
C04463=1008.051,320.462,343.731,169.473,53.827,160.444
C04464=1008.057,320.710,343.699,169.479,53.822,160.444
C04465=1008.062,320.958,343.667,169.487,53.816,160.444
C04466=1008.068,321.206,343.635,169.495,53.811,160.444
C04467=1008.073,321.454,343.603,169.502,53.804,160.445
C04468=1008.079,321.702,343.570,169.509,53.799,160.445
C04469=1008.085,321.950,343.538,169.516,53.793,160.445
C04470=1008.090,322.197,343.506,169.524,53.788,160.445
C04471=1008.096,322.445,343.474,169.531,53.782,160.445
C04472=1008.102,322.693,343.441,169.539,53.776,160.446
C04473=1008.107,322.941,343.409,169.546,53.770,160.446
C04474=1008.113,323.189,343.377,169.554,53.765,160.446
C04475=1008.120,323.437,343.344,169.560,53.759,160.447
C04476=1008.128,323.780,343.300,169.571,53.751,160.447
C04477=1008.135,324.125,343.255,169.581,53.743,160.447
C04478=1008.143,324.469,343.210,169.591,53.736,160.448
C04479=1008.152,324.812,343.165,169.603,53.728,160.448
C04480=1008.157,325.060,343.132,169.609,53.723,160.449
C04481=1008.163,325.309,343.099,169.617,53.717,160.449
C04482=1008.169,325.556,343.067,169.625,53.712,160.449
C04483=1008.174,325.803,343.034,169.632,53.706,160.450
C04484=1008.180,326.051,343.001,169.640,53.700,160.450
C04485=1008.186,326.299,342.967,169.647,53.695,160.450
C04486=1008.191,326.547,342.934,169.654,53.690,160.450
C04487=1008.197,326.795,342.902,169.662,53.684,160.451
C04488=1008.202,327.042,342.869,169.669,53.678,160.451
C04489=1008.208,327.290,342.836,169.677,53.673,160.451
C04490=1008.214,327.538,342.803,169.685,53.667,160.452
C04491=1008.220,327.786,342.770,169.692,53.662,160.452
C04492=1008.225,328.034,342.736,169.700,53.657,160.452
C04493=1008.231,328.281,342.704,169.707,53.651,160.453
C04494=1008.237,328.529,342.670,169.715,53.646,160.453
C04495=1008.243,328.777,342.638,169.722,53.640,160.453
C04496=1008.249,329.025,342.604,169.730,53.635,160.454
C04497=1008.254,329.272,342.571,169.738,53.630,160.454
C04498=1008.261,329.520,342.538,169.746,53.624,160.454
C04499=1008.267,329.767,342.504,169.753,53.618,160.455
C04500=1008.272,330.015,342.471,169.761,53.613,160.455
C04501=1008.278,330.263,342.438,169.768,53.608,160.456
C04502=1008.284,330.511,342.405,169.776,53.603,160.456
C04503=1008.290,330.758,342.372,169.783,53.597,160.456
C04504=1008.296,331.006,342.338,169.791,53.592,160.457
C04505=1008.302,331.253,342.305,169.799,53.587,160.457
C04506=1008.307,331.501,342.271,169.807,53.582,160.458
C04507=1008.313,331.749,342.237,169.815,53.576,160.458
C04508=1008.319,331.996,342.204,169.822,53.570,160.458
C04509=1008.325,332.244,342.170,169.830,53.566,160.459
C04510=1008.331,332.492,342.137,169.838,53.560,160.459
C04511=1008.337,332.739,342.103,169.846,53.555,160.460
C04512=1008.343,332.987,342.069,169.853,53.550,160.460
C04513=1008.349,333.235,342.035,169.861,53.545,160.460
C04514=1008.354,333.483,342.002,169.869,53.539,160.461
C04515=1008.360,333.730,341.968,169.877,53.534,160.461
C04516=1008.366,333.978,341.934,169.884,53.529,160.461
C04517=1008.372,334.226,341.900,169.892,53.524,160.462
C04518=1008.379,334.473,341.867,169.900,53.518,160.462
C04519=1008.384,334.721,341.833,169.908,53.513,160.463
C04520=1008.391,334.969,341.799,169.916,53.508,160.463
C04521=1008.397,335.216,341.765,169.924,53.503,160.464
C04522=1008.402,335.463,341.731,169.932,53.498,160.464
C04523=1008.409,335.712,341.697,169.940,53.493,160.465
C04524=1008.414,335.959,341.663,169.948,53.487,160.465
C04525=1008.420,336.206,341.629,169.956,53.482,160.465
C04526=1008.427,336.454,341.595,169.964,53.478,160.466
C04527=1008.433,336.701,341.561,169.971,53.472,160.466
C04528=1008.439,336.949,341.528,169.980,53.467,160.467
C04529=1008.445,337.197,341.493,169.988,53.462,160.467
C04530=1008.451,337.444,341.459,169.996,53.457,160.468
C04531=1008.458,337.692,341.425,170.003,53.452,160.468
C04532=1008.464,337.940,341.391,170.012,53.447,160.469
C04533=1008.469,338.187,341.357,170.020,53.442,160.469
C04534=1008.476,338.434,341.322,170.028,53.437,160.470
C04535=1008.481,338.682,341.287,170.036,53.432,160.470
C04536=1008.490,339.022,341.240,170.046,53.425,160.471
C04537=1008.498,339.361,341.193,170.057,53.418,160.472
C04538=1008.507,339.701,341.145,170.069,53.411,160.472
C04539=1008.516,340.041,341.098,170.079,53.405,160.473
C04540=1008.521,340.288,341.064,170.087,53.400,160.473
C04541=1008.528,340.535,341.029,170.096,53.395,160.474
C04542=1008.533,340.783,340.994,170.104,53.390,160.474
C04543=1008.540,341.031,340.960,170.112,53.385,160.475
C04544=1008.547,341.278,340.925,170.120,53.381,160.476
C04545=1008.552,341.526,340.891,170.128,53.376,160.476
C04546=1008.559,341.773,340.856,170.137,53.371,160.477
C04547=1008.565,342.021,340.821,170.145,53.366,160.477
C04548=1008.571,342.268,340.786,170.153,53.361,160.478
C04549=1008.578,342.516,340.751,170.161,53.356,160.478
C04550=1008.584,342.763,340.716,170.170,53.351,160.479
C04551=1008.589,343.011,340.682,170.178,53.346,160.479
C04552=1008.596,343.258,340.646,170.187,53.342,160.480
C04553=1008.603,343.506,340.611,170.195,53.337,160.481
C04554=1008.609,343.754,340.577,170.203,53.332,160.481
C04555=1008.616,344.000,340.542,170.211,53.327,160.482
C04556=1008.622,344.248,340.506,170.219,53.322,160.482
C04557=1008.628,344.496,340.472,170.228,53.318,160.483
C04558=1008.635,344.743,340.437,170.236,53.313,160.484
C04559=1008.642,344.991,340.402,170.244,53.308,160.484
C04560=1008.647,345.238,340.366,170.252,53.304,160.485
C04561=1008.654,345.485,340.331,170.261,53.298,160.485
C04562=1008.661,345.732,340.296,170.269,53.293,160.486
C04563=1008.667,345.980,340.260,170.278,53.289,160.487
C04564=1008.673,346.227,340.225,170.286,53.284,160.487
C04565=1008.680,346.475,340.190,170.295,53.280,160.488
C04566=1008.686,346.722,340.154,170.303,53.275,160.489
C04567=1008.693,346.970,340.119,170.311,53.271,160.489
C04568=1008.699,347.218,340.083,170.319,53.266,160.490
C04569=1008.706,347.465,340.048,170.329,53.261,160.491
C04570=1008.711,347.712,340.013,170.337,53.256,160.491
C04571=1008.718,347.959,339.978,170.346,53.252,160.492
C04572=1008.724,348.207,339.942,170.354,53.247,160.492
C04573=1008.732,348.454,339.906,170.362,53.243,160.493
C04574=1008.738,348.702,339.870,170.370,53.238,160.494
C04575=1008.745,348.949,339.835,170.380,53.234,160.494
C04576=1008.751,349.197,339.799,170.388,53.229,160.495
C04577=1008.758,349.444,339.763,170.397,53.224,160.496
C04578=1008.764,349.691,339.728,170.405,53.220,160.496
C04579=1008.771,349.938,339.692,170.414,53.216,160.497
C04580=1008.777,350.186,339.656,170.422,53.211,160.498
C04581=1008.784,350.433,339.621,170.431,53.206,160.499
C04582=1008.790,350.680,339.585,170.440,53.202,160.499
C04583=1008.797,350.928,339.549,170.448,53.198,160.500
C04584=1008.804,351.175,339.513,170.456,53.193,160.501
C04585=1008.810,351.423,339.477,170.466,53.188,160.501
C04586=1008.817,351.670,339.441,170.475,53.184,160.502
C04587=1008.823,351.917,339.406,170.483,53.180,160.503
C04588=1008.831,352.165,339.370,170.492,53.176,160.504
C04589=1008.837,352.412,339.333,170.500,53.171,160.504
C04590=1008.843,352.659,339.297,170.509,53.166,160.505
C04591=1008.851,352.906,339.262,170.518,53.162,160.506
C04592=1008.857,353.154,339.225,170.526,53.158,160.506
C04593=1008.864,353.401,339.188,170.535,53.153,160.507
C04594=1008.870,353.648,339.152,170.544,53.149,160.508
C04595=1008.878,353.896,339.116,170.553,53.145,160.509
C04596=1008.885,354.194,339.072,170.564,53.140,160.510
C04597=1008.894,354.493,339.029,170.574,53.134,160.511
C04598=1008.902,354.792,338.984,170.586,53.129,160.512
C04599=1008.910,355.090,338.940,170.596,53.124,160.513
C04600=1008.918,355.338,338.904,170.605,53.120,160.513
C04601=1008.924,355.585,338.867,170.613,53.116,160.514
C04602=1008.931,355.832,338.830,170.623,53.111,160.515
C04603=1008.938,356.079,338.795,170.631,53.107,160.516
C04604=1008.945,356.327,338.758,170.640,53.103,160.517
C04605=1008.951,356.574,338.721,170.650,53.098,160.517
C04606=1008.958,356.822,338.685,170.658,53.094,160.518
C04607=1008.965,357.068,338.649,170.667,53.090,160.519
C04608=1008.642,354.940,338.607,170.571,53.176,160.520
C04609=1008.636,354.694,338.642,170.563,53.180,160.520
C04610=1008.628,354.447,338.678,170.553,53.185,160.519
C04611=1008.622,354.202,338.715,170.545,53.189,160.518
C04612=1008.615,353.955,338.751,170.536,53.194,160.517
C04613=1008.608,353.708,338.786,170.527,53.198,160.517
C04614=1008.601,353.461,338.823,170.518,53.202,160.516
C04615=1008.595,353.213,338.860,170.509,53.207,160.515
C04616=1008.589,352.966,338.895,170.501,53.211,160.514
C04617=1008.581,352.718,338.932,170.491,53.216,160.513
C04618=1008.575,352.471,338.968,170.483,53.220,160.513
C04619=1008.569,352.224,339.004,170.474,53.224,160.512
C04620=1008.562,351.977,339.040,170.466,53.228,160.511
C04621=1008.556,351.730,339.076,170.456,53.233,160.510
C04622=1008.548,351.482,339.112,170.448,53.237,160.510
C04623=1008.541,351.235,339.148,170.440,53.242,160.509
C04624=1008.535,350.987,339.183,170.431,53.246,160.508
C04625=1008.528,350.740,339.218,170.422,53.251,160.508
C04626=1008.522,350.493,339.255,170.413,53.255,160.507
C04627=1008.515,350.246,339.290,170.405,53.260,160.506
C04628=1008.508,349.998,339.327,170.396,53.264,160.506
C04629=1008.501,349.750,339.362,170.388,53.269,160.505
C04630=1008.495,349.503,339.398,170.379,53.273,160.504
C04631=1008.488,349.256,339.433,170.370,53.278,160.503
C04632=1008.482,349.008,339.469,170.361,53.282,160.503
C04633=1008.476,348.761,339.504,170.353,53.287,160.502
C04634=1008.470,348.513,339.540,170.345,53.292,160.501
C04635=1008.463,348.266,339.575,170.336,53.296,160.501
C04636=1008.456,348.019,339.612,170.328,53.300,160.500
C04637=1008.450,347.772,339.647,170.319,53.305,160.499
C04638=1008.444,347.524,339.683,170.310,53.310,160.499
C04639=1008.437,347.276,339.718,170.302,53.315,160.498
C04640=1008.431,347.029,339.753,170.293,53.319,160.497
C04641=1008.425,346.782,339.788,170.285,53.324,160.497
C04642=1008.419,346.534,339.824,170.277,53.328,160.496
C04643=1008.412,346.287,339.859,170.269,53.333,160.495
C04644=1008.405,346.040,339.894,170.259,53.338,160.495
C04645=1008.399,345.792,339.930,170.251,53.342,160.494
C04646=1008.392,345.545,339.965,170.242,53.347,160.493
C04647=1008.386,345.297,340.001,170.234,53.352,160.493
C04648=1008.380,345.050,340.035,170.226,53.357,160.492
C04649=1008.374,344.802,340.070,170.218,53.361,160.492
C04650=1008.367,344.555,340.105,170.210,53.366,160.491
C04651=1008.361,344.307,340.141,170.202,53.371,160.491
C04652=1008.354,344.059,340.175,170.193,53.375,160.490
C04653=1008.348,343.813,340.210,170.184,53.380,160.489
C04654=1008.341,343.565,340.245,170.176,53.385,160.489
C04655=1008.335,343.317,340.280,170.168,53.390,160.488
C04656=1008.330,343.070,340.315,170.159,53.394,160.487
C04657=1008.323,342.822,340.349,170.151,53.399,160.487
C04658=1008.316,342.575,340.384,170.143,53.404,160.486
C04659=1008.310,342.327,340.419,170.135,53.409,160.486
C04660=1008.304,342.080,340.454,170.127,53.414,160.485
C04661=1008.298,341.832,340.489,170.119,53.419,160.485
C04662=1008.292,341.585,340.523,170.110,53.423,160.484
C04663=1008.285,341.337,340.558,170.102,53.428,160.483
C04664=1008.279,341.089,340.592,170.094,53.433,160.483
C04665=1008.273,340.842,340.628,170.086,53.438,160.482
C04666=1008.267,340.594,340.662,170.078,53.443,160.482
C04667=1008.261,340.347,340.696,170.070,53.448,160.481
C04668=1008.254,340.100,340.731,170.062,53.453,160.481
C04669=1008.246,339.758,340.779,170.050,53.460,160.480
C04670=1008.237,339.416,340.826,170.039,53.467,160.479
C04671=1008.229,339.074,340.874,170.027,53.473,160.478
C04672=1008.221,338.732,340.921,170.016,53.480,160.478
C04673=1008.214,338.484,340.956,170.008,53.485,160.477
C04674=1008.209,338.237,340.990,170.000,53.490,160.477
C04675=1008.203,337.990,341.024,169.993,53.495,160.476
C04676=1008.197,337.741,341.059,169.985,53.500,160.476
C04677=1008.191,337.494,341.093,169.976,53.505,160.475
C04678=1008.185,337.246,341.127,169.968,53.510,160.475
C04679=1008.179,336.999,341.161,169.960,53.515,160.474
C04680=1008.172,336.752,341.195,169.953,53.521,160.474
C04681=1008.166,336.504,341.229,169.945,53.526,160.473
C04682=1008.160,336.257,341.263,169.936,53.530,160.473
C04683=1008.154,336.009,341.296,169.928,53.535,160.472
C04684=1008.148,335.761,341.331,169.921,53.541,160.472
C04685=1008.142,335.513,341.365,169.913,53.546,160.472
C04686=1008.136,335.266,341.398,169.904,53.551,160.471
C04687=1008.131,335.018,341.432,169.896,53.556,160.470
C04688=1008.124,334.770,341.467,169.889,53.561,160.470
C04689=1008.118,334.523,341.499,169.881,53.566,160.470
C04690=1008.112,334.275,341.534,169.873,53.572,160.469
C04691=1008.106,334.028,341.568,169.866,53.576,160.469
C04692=1008.100,333.780,341.601,169.858,53.581,160.468
C04693=1008.094,333.532,341.635,169.850,53.587,160.468
C04694=1008.089,333.284,341.669,169.842,53.592,160.467
C04695=1008.083,333.037,341.703,169.834,53.597,160.467
C04696=1008.077,332.789,341.736,169.826,53.602,160.467
C04697=1008.071,332.542,341.770,169.819,53.608,160.466
C04698=1008.065,332.294,341.803,169.811,53.613,160.466
C04699=1008.059,332.047,341.837,169.803,53.619,160.465
C04700=1008.053,331.798,341.871,169.795,53.623,160.465
C04701=1008.047,331.550,341.904,169.787,53.629,160.465
C04702=1008.042,331.303,341.938,169.780,53.634,160.464
C04703=1008.036,331.055,341.971,169.773,53.639,160.464
C04704=1008.030,330.808,342.004,169.764,53.644,160.463
C04705=1008.024,330.560,342.037,169.757,53.650,160.463
C04706=1008.018,330.313,342.071,169.749,53.655,160.463
C04707=1008.012,330.065,342.104,169.741,53.660,160.462
C04708=1008.006,329.817,342.138,169.733,53.666,160.462
C04709=1008.001,329.569,342.171,169.726,53.672,160.462
C04710=1007.995,329.322,342.204,169.718,53.676,160.461
C04711=1007.989,329.074,342.237,169.710,53.682,160.461
C04712=1007.983,328.826,342.270,169.703,53.687,160.460
C04713=1007.977,328.578,342.303,169.696,53.693,160.460
C04714=1007.972,328.331,342.336,169.688,53.698,160.460
C04715=1007.966,328.083,342.369,169.680,53.703,160.459
C04716=1007.960,327.835,342.402,169.672,53.709,160.459
C04717=1007.955,327.588,342.435,169.665,53.715,160.459
C04718=1007.949,327.340,342.468,169.657,53.720,160.458
C04719=1007.943,327.092,342.502,169.650,53.725,160.458
C04720=1007.938,326.843,342.534,169.642,53.730,160.458
C04721=1007.932,326.597,342.567,169.635,53.736,160.457
C04722=1007.927,326.349,342.600,169.627,53.742,160.457
C04723=1007.920,326.101,342.633,169.620,53.747,160.457
C04724=1007.915,325.853,342.666,169.612,53.753,160.456
C04725=1007.909,325.605,342.699,169.605,53.758,160.456
C04726=1007.904,325.358,342.731,169.597,53.763,160.456
C04727=1007.898,325.110,342.764,169.590,53.769,160.455
C04728=1007.893,324.862,342.798,169.582,53.774,160.455
C04729=1007.884,324.515,342.842,169.572,53.783,160.455
C04730=1007.876,324.169,342.888,169.561,53.790,160.454
C04731=1007.868,323.823,342.932,169.551,53.798,160.454
C04732=1007.860,323.477,342.978,169.541,53.805,160.453
C04733=1007.855,323.229,343.010,169.533,53.811,160.453
C04734=1007.849,322.981,343.042,169.526,53.817,160.453
C04735=1007.843,322.734,343.075,169.518,53.823,160.453
C04736=1007.837,322.486,343.107,169.511,53.829,160.452
C04737=1007.831,322.237,343.139,169.504,53.834,160.452
C04738=1007.826,321.990,343.171,169.496,53.839,160.452
C04739=1007.820,321.742,343.204,169.489,53.845,160.451
C04740=1007.815,321.494,343.235,169.481,53.851,160.451
C04741=1007.809,321.246,343.267,169.474,53.857,160.451
C04742=1007.803,320.999,343.299,169.467,53.862,160.451
C04743=1007.797,320.751,343.331,169.460,53.868,160.450
C04744=1007.792,320.503,343.364,169.452,53.874,160.450
C04745=1007.786,320.255,343.396,169.445,53.880,160.450
C04746=1007.780,320.007,343.428,169.437,53.885,160.450
C04747=1007.775,319.759,343.460,169.431,53.891,160.449
C04748=1007.770,319.512,343.491,169.423,53.896,160.449
C04749=1007.764,319.264,343.523,169.416,53.903,160.449
C04750=1007.759,319.016,343.556,169.408,53.908,160.449
C04751=1007.753,318.768,343.588,169.402,53.914,160.448
C04752=1007.748,318.520,343.619,169.395,53.920,160.448
C04753=1007.742,318.272,343.651,169.387,53.925,160.448
C04754=1007.736,318.024,343.683,169.379,53.931,160.448
C04755=1007.732,317.777,343.715,169.373,53.937,160.448
C04756=1007.726,317.528,343.747,169.365,53.943,160.447
C04757=1007.721,317.280,343.778,169.358,53.948,160.447
C04758=1007.715,317.033,343.810,169.351,53.955,160.447
C04759=1007.709,316.784,343.842,169.344,53.960,160.447
C04760=1007.704,316.537,343.874,169.337,53.966,160.447
C04761=1007.699,316.289,343.906,169.329,53.972,160.446
C04762=1007.693,316.041,343.938,169.322,53.978,160.446
C04763=1007.688,315.793,343.969,169.315,53.983,160.446
C04764=1007.683,315.545,344.000,169.308,53.990,160.446
C04765=1007.677,315.298,344.032,169.301,53.995,160.445
C04766=1007.672,315.049,344.063,169.295,54.001,160.445
C04767=1007.667,314.801,344.096,169.287,54.007,160.445
C04768=1007.662,314.554,344.127,169.280,54.013,160.445
C04769=1007.656,314.306,344.159,169.272,54.019,160.445
C04770=1007.651,314.058,344.190,169.266,54.025,160.445
C04771=1007.646,313.810,344.222,169.258,54.030,160.444
C04772=1007.640,313.562,344.253,169.251,54.037,160.444
C04773=1007.635,313.314,344.285,169.245,54.042,160.444
C04774=1007.630,313.066,344.317,169.237,54.048,160.444
C04775=1007.625,312.818,344.348,169.230,54.055,160.444
C04776=1007.620,312.571,344.379,169.224,54.060,160.444
C04777=1007.614,312.323,344.410,169.217,54.066,160.443
C04778=1007.609,312.075,344.442,169.209,54.073,160.443
C04779=1007.605,311.827,344.474,169.203,54.078,160.443
C04780=1007.599,311.579,344.505,169.196,54.084,160.443
C04781=1007.594,311.331,344.536,169.188,54.091,160.443
C04782=1007.589,311.083,344.567,169.182,54.096,160.443
C04783=1007.584,310.835,344.599,169.175,54.102,160.443
C04784=1007.579,310.587,344.630,169.168,54.109,160.442
C04785=1007.574,310.339,344.662,169.161,54.114,160.442
C04786=1007.569,310.091,344.693,169.154,54.120,160.442
C04787=1007.564,309.843,344.724,169.148,54.126,160.442
C04788=1007.559,309.596,344.756,169.140,54.132,160.442
C04789=1007.552,309.255,344.798,169.131,54.141,160.442
C04790=1007.545,308.915,344.841,169.121,54.149,160.441
C04791=1007.538,308.573,344.884,169.111,54.157,160.441
C04792=1007.531,308.233,344.927,169.103,54.166,160.441
C04793=1007.527,307.986,344.957,169.096,54.171,160.441
C04794=1007.521,307.738,344.988,169.088,54.178,160.441
C04795=1007.515,307.490,345.018,169.082,54.184,160.441
C04796=1007.510,307.242,345.049,169.075,54.190,160.441
C04797=1007.505,306.993,345.079,169.068,54.196,160.441
C04798=1007.500,306.746,345.109,169.062,54.202,160.441
C04799=1007.494,306.498,345.140,169.055,54.209,160.441
C04800=1007.489,306.250,345.171,169.048,54.215,160.440
C04801=1007.484,306.001,345.200,169.041,54.221,160.440
C04802=1007.479,305.753,345.231,169.034,54.227,160.440
C04803=1007.474,305.505,345.262,169.027,54.234,160.440
C04804=1007.469,305.257,345.291,169.021,54.240,160.440
C04805=1007.464,305.009,345.322,169.014,54.246,160.440
C04806=1007.458,304.762,345.353,169.007,54.252,160.440
C04807=1007.453,304.513,345.383,169.001,54.258,160.440
C04808=1007.448,304.266,345.413,168.993,54.265,160.440
C04809=1007.443,304.017,345.443,168.986,54.271,160.440
C04810=1007.437,303.769,345.474,168.980,54.277,160.440
C04811=1007.432,303.521,345.504,168.973,54.283,160.439
C04812=1007.427,303.273,345.534,168.966,54.290,160.440
C04813=1007.420,302.912,345.578,168.957,54.299,160.440
C04814=1007.412,302.550,345.622,168.947,54.309,160.439
C04815=1007.404,302.189,345.666,168.938,54.318,160.439
C04816=1007.397,301.828,345.710,168.928,54.327,160.439
C04817=1007.155,302.488,345.264,168.923,54.352,160.444
C04818=1007.159,302.715,345.236,168.930,54.346,160.444
C04819=1007.163,302.940,345.209,168.936,54.340,160.444
C04820=1007.169,303.166,345.181,168.942,54.334,160.444
C04821=1007.173,303.391,345.154,168.948,54.329,160.444
C04822=1007.177,303.618,345.126,168.954,54.324,160.444
C04823=1007.182,303.844,345.099,168.960,54.318,160.445
C04824=1007.187,304.069,345.072,168.967,54.312,160.445
C04825=1007.191,304.296,345.044,168.973,54.306,160.445
C04826=1007.197,304.544,345.014,168.979,54.300,160.445
C04827=1007.201,304.793,344.983,168.986,54.294,160.445
C04828=1007.207,305.040,344.953,168.993,54.288,160.445
C04829=1007.211,305.288,344.923,168.999,54.282,160.445
C04830=1007.217,305.536,344.893,169.007,54.275,160.445
C04831=1007.222,305.784,344.862,169.013,54.269,160.445
C04832=1007.227,306.032,344.833,169.020,54.263,160.445
C04833=1007.232,306.280,344.802,169.027,54.257,160.445
C04834=1007.238,306.528,344.771,169.033,54.251,160.445
C04835=1007.243,306.777,344.741,169.041,54.245,160.446
C04836=1007.249,307.025,344.711,169.048,54.239,160.446
C04837=1007.254,307.273,344.680,169.054,54.233,160.446
C04838=1007.259,307.520,344.650,169.061,54.226,160.446
C04839=1007.264,307.768,344.619,169.068,54.220,160.446
C04840=1007.270,308.016,344.589,169.075,54.214,160.446
C04841=1007.275,308.265,344.558,169.082,54.208,160.446
C04842=1007.281,308.607,344.515,169.091,54.199,160.447
C04843=1007.288,308.949,344.472,169.101,54.191,160.447
C04844=1007.295,309.292,344.429,169.111,54.183,160.447
C04845=1007.302,309.635,344.386,169.119,54.175,160.447
C04846=1007.307,309.883,344.355,169.127,54.169,160.447
C04847=1007.312,310.131,344.324,169.134,54.162,160.447
C04848=1007.317,310.380,344.292,169.140,54.157,160.448
C04849=1007.322,310.627,344.261,169.148,54.151,160.448
C04850=1007.327,310.875,344.230,169.155,54.144,160.448
C04851=1007.332,311.123,344.199,169.161,54.139,160.448
C04852=1007.338,311.371,344.167,169.168,54.133,160.448
C04853=1007.342,311.619,344.135,169.175,54.127,160.448
C04854=1007.347,311.867,344.104,169.182,54.121,160.449
C04855=1007.352,312.115,344.073,169.189,54.115,160.449
C04856=1007.358,312.362,344.041,169.196,54.110,160.449
C04857=1007.363,312.611,344.010,169.203,54.103,160.449
C04858=1007.368,312.859,343.979,169.211,54.098,160.449
C04859=1007.373,313.107,343.947,169.217,54.092,160.449
C04860=1007.378,313.354,343.915,169.225,54.086,160.450
C04861=1007.383,313.602,343.884,169.232,54.080,160.450
C04862=1007.388,313.850,343.853,169.238,54.074,160.450
C04863=1007.393,314.098,343.822,169.245,54.068,160.450
C04864=1007.399,314.345,343.790,169.253,54.062,160.450
C04865=1007.403,314.594,343.759,169.259,54.056,160.451
C04866=1007.409,314.842,343.727,169.267,54.051,160.451
C04867=1007.415,315.090,343.695,169.274,54.044,160.451
C04868=1007.420,315.338,343.664,169.281,54.039,160.451
C04869=1007.425,315.585,343.632,169.288,54.033,160.451
C04870=1007.430,315.833,343.601,169.295,54.027,160.452
C04871=1007.435,316.082,343.569,169.303,54.021,160.452
C04872=1007.441,316.329,343.537,169.309,54.016,160.452
C04873=1007.446,316.577,343.505,169.317,54.010,160.452
C04874=1007.452,316.824,343.474,169.324,54.004,160.452
C04875=1007.458,317.073,343.442,169.331,53.998,160.453
C04876=1007.463,317.321,343.411,169.338,53.993,160.453
C04877=1007.467,317.569,343.379,169.345,53.986,160.453
C04878=1007.473,317.817,343.347,169.353,53.981,160.454
C04879=1007.479,318.064,343.315,169.360,53.975,160.454
C04880=1007.484,318.312,343.283,169.367,53.969,160.454
C04881=1007.490,318.560,343.251,169.374,53.964,160.454
C04882=1007.495,318.807,343.220,169.382,53.958,160.455
C04883=1007.500,319.055,343.187,169.388,53.952,160.454
C04884=1007.506,319.304,343.155,169.396,53.946,160.455
C04885=1007.511,319.551,343.124,169.403,53.941,160.455
C04886=1007.517,319.799,343.092,169.411,53.935,160.456
C04887=1007.523,320.047,343.060,169.418,53.930,160.456
C04888=1007.528,320.295,343.027,169.425,53.923,160.456
C04889=1007.533,320.543,342.996,169.432,53.918,160.456
C04890=1007.539,320.791,342.964,169.440,53.912,160.457
C04891=1007.545,321.039,342.932,169.447,53.907,160.457
C04892=1007.551,321.287,342.900,169.454,53.901,160.457
C04893=1007.556,321.534,342.868,169.462,53.896,160.457
C04894=1007.561,321.783,342.836,169.469,53.889,160.457
C04895=1007.567,322.030,342.804,169.477,53.884,160.458
C04896=1007.573,322.278,342.771,169.483,53.878,160.458
C04897=1007.579,322.526,342.739,169.491,53.873,160.458
C04898=1007.584,322.774,342.708,169.499,53.867,160.459
C04899=1007.590,323.022,342.676,169.506,53.862,160.459
C04900=1007.595,323.269,342.643,169.514,53.856,160.459
C04901=1007.601,323.517,342.611,169.521,53.851,160.460
C04902=1007.610,323.866,342.565,169.532,53.843,160.460
C04903=1007.617,324.215,342.520,169.542,53.835,160.461
C04904=1007.626,324.563,342.474,169.553,53.827,160.461
C04905=1007.634,324.912,342.429,169.563,53.819,160.461
C04906=1007.639,325.159,342.396,169.570,53.814,160.462
C04907=1007.645,325.408,342.363,169.578,53.808,160.462
C04908=1007.651,325.655,342.331,169.585,53.803,160.462
C04909=1007.656,325.902,342.298,169.593,53.798,160.463
C04910=1007.661,326.150,342.264,169.600,53.792,160.463
C04911=1007.667,326.398,342.232,169.608,53.787,160.463
C04912=1007.673,326.646,342.199,169.616,53.781,160.464
C04913=1007.679,326.893,342.166,169.623,53.775,160.464
C04914=1007.684,327.141,342.133,169.630,53.771,160.465
C04915=1007.690,327.389,342.100,169.638,53.765,160.465
C04916=1007.696,327.637,342.068,169.646,53.759,160.465
C04917=1007.701,327.885,342.034,169.653,53.754,160.465
C04918=1007.707,328.133,342.001,169.661,53.749,160.466
C04919=1007.713,328.380,341.969,169.669,53.743,160.466
C04920=1007.718,328.628,341.935,169.676,53.738,160.467
C04921=1007.724,328.876,341.903,169.684,53.733,160.467
C04922=1007.730,329.123,341.869,169.691,53.727,160.467
C04923=1007.735,329.371,341.836,169.699,53.722,160.468
C04924=1007.742,329.619,341.803,169.707,53.717,160.468
C04925=1007.747,329.867,341.770,169.715,53.711,160.469
C04926=1007.753,330.115,341.737,169.722,53.706,160.469
C04927=1007.759,330.362,341.704,169.730,53.701,160.470
C04928=1007.765,330.610,341.670,169.737,53.696,160.470
C04929=1007.770,330.858,341.637,169.745,53.691,160.470
C04930=1007.777,331.105,341.604,169.753,53.685,160.471
C04931=1007.782,331.353,341.570,169.760,53.679,160.471
C04932=1007.788,331.601,341.537,169.769,53.674,160.471
C04933=1007.794,331.848,341.503,169.776,53.669,160.472
C04934=1007.799,332.096,341.470,169.784,53.664,160.472
C04935=1007.805,332.344,341.436,169.792,53.659,160.473
C04936=1007.811,332.591,341.402,169.800,53.653,160.473
C04937=1007.817,332.839,341.369,169.807,53.649,160.474
C04938=1007.823,333.086,341.335,169.815,53.643,160.474
C04939=1007.829,333.334,341.302,169.823,53.638,160.474
C04940=1007.835,333.582,341.268,169.830,53.633,160.475
C04941=1007.841,333.830,341.234,169.839,53.628,160.475
C04942=1007.846,334.077,341.200,169.847,53.623,160.476
C04943=1007.852,334.325,341.167,169.854,53.617,160.476
C04944=1007.858,334.572,341.133,169.862,53.612,160.477
C04945=1007.863,334.820,341.100,169.871,53.607,160.477
C04946=1007.871,335.068,341.066,169.878,53.602,160.478
C04947=1007.876,335.315,341.032,169.886,53.597,160.478
C04948=1007.882,335.563,340.998,169.894,53.592,160.479
C04949=1007.888,335.810,340.964,169.902,53.587,160.479
C04950=1007.894,336.058,340.930,169.910,53.581,160.480
C04951=1007.900,336.306,340.897,169.918,53.576,160.480
C04952=1007.906,336.554,340.862,169.926,53.571,160.481
C04953=1007.912,336.802,340.828,169.933,53.567,160.481
C04954=1007.918,337.049,340.794,169.941,53.562,160.482
C04955=1007.924,337.296,340.761,169.949,53.556,160.482
C04956=1007.931,337.544,340.727,169.957,53.551,160.482
C04957=1007.936,337.792,340.692,169.965,53.546,160.483
C04958=1007.942,338.039,340.658,169.973,53.542,160.484
C04959=1007.948,338.287,340.624,169.981,53.537,160.484
C04960=1007.954,338.535,340.590,169.990,53.532,160.485
C04961=1007.961,338.782,340.555,169.998,53.527,160.485
C04962=1007.968,339.072,340.515,170.008,53.521,160.486
C04963=1007.974,339.363,340.474,170.016,53.515,160.486
C04964=1007.982,339.653,340.434,170.027,53.509,160.487
C04965=1007.989,339.943,340.394,170.037,53.504,160.488
C04966=1007.995,340.190,340.359,170.045,53.499,160.488
C04967=1008.001,340.438,340.324,170.053,53.494,160.489
C04968=1008.007,340.685,340.290,170.061,53.489,160.489
C04969=1008.013,340.933,340.256,170.069,53.484,160.490
C04970=1008.020,341.180,340.221,170.077,53.479,160.490
C04971=1008.026,341.428,340.187,170.085,53.474,160.491
C04972=1008.031,341.675,340.152,170.093,53.469,160.492
C04973=1008.038,341.923,340.117,170.101,53.464,160.492
C04974=1008.044,342.171,340.083,170.110,53.460,160.493
C04975=1008.051,342.417,340.048,170.118,53.455,160.493
C04976=1008.057,342.665,340.013,170.126,53.450,160.494
C04977=1008.063,342.913,339.978,170.134,53.445,160.494
C04978=1008.069,343.160,339.944,170.143,53.441,160.495
C04979=1008.076,343.408,339.908,170.151,53.436,160.496
C04980=1008.082,343.656,339.874,170.159,53.431,160.496
C04981=1008.088,343.903,339.839,170.167,53.426,160.497
C04982=1008.094,344.151,339.804,170.176,53.422,160.498
C04983=1008.101,344.398,339.769,170.185,53.417,160.498
C04984=1008.108,344.645,339.734,170.193,53.412,160.499
C04985=1008.113,344.893,339.700,170.201,53.407,160.499
C04986=1008.119,345.140,339.664,170.209,53.402,160.500
C04987=1008.126,345.388,339.629,170.218,53.398,160.501
C04988=1008.133,345.635,339.594,170.226,53.393,160.501
C04989=1008.139,345.883,339.558,170.234,53.388,160.502
C04990=1008.145,346.129,339.523,170.243,53.384,160.503
C04991=1008.151,346.378,339.488,170.251,53.379,160.503
C04992=1008.158,346.625,339.453,170.260,53.374,160.504
C04993=1008.164,346.873,339.418,170.269,53.370,160.504
C04994=1008.170,347.120,339.382,170.277,53.365,160.505
C04995=1008.177,347.367,339.347,170.286,53.361,160.506
C04996=1008.183,347.615,339.312,170.294,53.356,160.507
C04997=1008.190,347.862,339.276,170.302,53.352,160.507
C04998=1008.196,348.109,339.240,170.310,53.347,160.508
C04999=1008.203,348.356,339.205,170.320,53.342,160.509
C05000=1008.209,348.604,339.169,170.329,53.338,160.509
C05001=1008.215,348.851,339.134,170.337,53.333,160.510
C05002=1008.221,349.099,339.099,170.345,53.329,160.511
C05003=1008.228,349.346,339.063,170.354,53.325,160.511
C05004=1008.234,349.593,339.027,170.362,53.320,160.512
C05005=1008.242,349.841,338.992,170.371,53.315,160.513
C05006=1008.248,350.089,338.956,170.380,53.311,160.514
C05007=1008.255,350.336,338.920,170.388,53.307,160.514
C05008=1008.261,350.583,338.884,170.397,53.302,160.515
C05009=1008.268,350.830,338.848,170.405,53.297,160.516
C05010=1008.274,351.078,338.813,170.415,53.293,160.516
C05011=1008.281,351.325,338.777,170.423,53.288,160.517
C05012=1008.287,351.572,338.741,170.432,53.284,160.518
C05013=1008.295,351.820,338.706,170.440,53.280,160.519
C05014=1008.301,352.067,338.669,170.450,53.275,160.520
C05015=1008.308,352.315,338.634,170.458,53.271,160.520
C05016=1008.314,352.562,338.598,170.467,53.267,160.521
C05017=1008.320,352.809,338.561,170.476,53.263,160.522
C05018=1008.000,350.672,338.514,170.381,53.347,160.523
C05019=1007.994,350.425,338.550,170.372,53.351,160.522
C05020=1007.988,350.177,338.585,170.364,53.356,160.521
C05021=1007.981,349.930,338.621,170.355,53.361,160.521
C05022=1007.975,349.683,338.656,170.346,53.365,160.520
C05023=1007.968,349.435,338.692,170.337,53.369,160.519
C05024=1007.962,349.188,338.727,170.329,53.374,160.518
C05025=1007.955,348.941,338.764,170.321,53.379,160.518
C05026=1007.949,348.693,338.799,170.312,53.383,160.517
C05027=1007.943,348.446,338.834,170.303,53.388,160.516
C05028=1007.936,348.198,338.870,170.294,53.392,160.515
C05029=1007.930,347.951,338.905,170.286,53.397,160.515
C05030=1007.923,347.703,338.940,170.278,53.401,160.514
C05031=1007.917,347.456,338.976,170.269,53.406,160.514
C05032=1007.910,347.208,339.011,170.261,53.410,160.513
C05033=1007.903,346.961,339.046,170.251,53.415,160.512
C05034=1007.897,346.713,339.082,170.243,53.420,160.511
C05035=1007.891,346.467,339.117,170.235,53.424,160.511
C05036=1007.885,346.219,339.153,170.227,53.429,160.510
C05037=1007.878,345.972,339.188,170.218,53.433,160.509
C05038=1007.872,345.724,339.224,170.210,53.438,160.509
C05039=1007.866,345.476,339.258,170.201,53.442,160.508
C05040=1007.860,345.229,339.293,170.193,53.447,160.508
C05041=1007.854,344.982,339.328,170.185,53.452,160.507
C05042=1007.847,344.734,339.363,170.176,53.457,160.506
C05043=1007.841,344.486,339.398,170.167,53.461,160.505
C05044=1007.834,344.240,339.433,170.159,53.466,160.505
C05045=1007.829,343.991,339.468,170.151,53.471,160.504
C05046=1007.822,343.744,339.503,170.142,53.475,160.503
C05047=1007.816,343.497,339.537,170.134,53.480,160.503
C05048=1007.809,343.249,339.572,170.126,53.485,160.502
C05049=1007.803,343.001,339.607,170.118,53.489,160.502
C05050=1007.797,342.754,339.642,170.109,53.494,160.501
C05051=1007.791,342.506,339.676,170.101,53.499,160.501
C05052=1007.785,342.260,339.711,170.093,53.504,160.500
C05053=1007.778,342.012,339.745,170.085,53.508,160.499
C05054=1007.773,341.763,339.780,170.077,53.513,160.499
C05055=1007.766,341.517,339.815,170.069,53.518,160.498
C05056=1007.760,341.269,339.850,170.060,53.523,160.498
C05057=1007.754,341.021,339.884,170.052,53.528,160.497
C05058=1007.747,340.774,339.919,170.043,53.534,160.497
C05059=1007.742,340.531,339.952,170.036,53.537,160.496
C05060=1007.736,340.289,339.986,170.028,53.542,160.495
C05061=1007.730,340.046,340.020,170.019,53.547,160.495
C05062=1007.724,339.802,340.054,170.011,53.552,160.494
C05063=1007.718,339.560,340.087,170.003,53.557,160.494
C05064=1007.712,339.318,340.121,169.995,53.562,160.493
C05065=1007.706,339.074,340.155,169.988,53.567,160.493
C05066=1007.701,338.832,340.189,169.980,53.572,160.492
C05067=1007.694,338.584,340.223,169.972,53.576,160.492
C05068=1007.688,338.337,340.257,169.964,53.581,160.491
C05069=1007.682,338.089,340.292,169.956,53.586,160.491
C05070=1007.676,337.842,340.326,169.948,53.591,160.490
C05071=1007.671,337.594,340.360,169.940,53.596,160.489
C05072=1007.664,337.346,340.395,169.931,53.601,160.489
C05073=1007.658,337.099,340.427,169.923,53.606,160.488
C05074=1007.652,336.851,340.461,169.915,53.611,160.488
C05075=1007.646,336.604,340.496,169.907,53.616,160.487
C05076=1007.640,336.356,340.530,169.899,53.621,160.487
C05077=1007.634,336.108,340.563,169.891,53.627,160.486
C05078=1007.628,335.861,340.597,169.883,53.631,160.486
C05079=1007.623,335.614,340.631,169.875,53.636,160.485
C05080=1007.616,335.365,340.665,169.867,53.641,160.485
C05081=1007.611,335.118,340.699,169.859,53.646,160.484
C05082=1007.604,334.870,340.732,169.851,53.652,160.484
C05083=1007.598,334.623,340.766,169.844,53.656,160.483
C05084=1007.593,334.375,340.799,169.836,53.661,160.483
C05085=1007.586,334.127,340.834,169.828,53.666,160.482
C05086=1007.581,333.879,340.867,169.820,53.672,160.482
C05087=1007.575,333.632,340.901,169.812,53.677,160.481
C05088=1007.569,333.384,340.934,169.804,53.682,160.481
C05089=1007.564,333.137,340.968,169.797,53.687,160.481
C05090=1007.558,332.889,341.002,169.788,53.692,160.480
C05091=1007.551,332.642,341.035,169.781,53.698,160.480
C05092=1007.546,332.394,341.069,169.773,53.703,160.479
C05093=1007.540,332.146,341.102,169.765,53.708,160.479
C05094=1007.534,331.899,341.136,169.758,53.713,160.478
C05095=1007.529,331.651,341.169,169.750,53.718,160.478
C05096=1007.523,331.403,341.203,169.742,53.724,160.478
C05097=1007.518,331.155,341.236,169.734,53.729,160.477
C05098=1007.512,330.908,341.270,169.727,53.734,160.477
C05099=1007.506,330.660,341.303,169.718,53.739,160.476
C05100=1007.500,330.412,341.336,169.711,53.745,160.476
C05101=1007.494,330.165,341.369,169.703,53.750,160.475
C05102=1007.488,329.917,341.402,169.696,53.755,160.475
C05103=1007.483,329.669,341.436,169.688,53.760,160.474
C05104=1007.476,329.421,341.468,169.680,53.766,160.474
C05105=1007.471,329.173,341.502,169.673,53.771,160.474
C05106=1007.465,328.925,341.535,169.665,53.776,160.473
C05107=1007.459,328.678,341.568,169.657,53.782,160.473
C05108=1007.454,328.431,341.601,169.649,53.787,160.473
C05109=1007.449,328.182,341.633,169.642,53.792,160.472
C05110=1007.442,327.934,341.666,169.635,53.798,160.472
C05111=1007.437,327.686,341.699,169.627,53.803,160.472
C05112=1007.431,327.439,341.732,169.619,53.808,160.471
C05113=1007.425,327.191,341.765,169.611,53.814,160.471
C05114=1007.420,326.944,341.798,169.605,53.819,160.470
C05115=1007.414,326.696,341.830,169.597,53.824,160.470
C05116=1007.409,326.448,341.864,169.589,53.830,160.470
C05117=1007.403,326.200,341.897,169.581,53.835,160.469
C05118=1007.398,325.952,341.929,169.574,53.841,160.469
C05119=1007.392,325.704,341.962,169.566,53.847,160.469
C05120=1007.386,325.456,341.996,169.559,53.851,160.468
C05121=1007.381,325.209,342.027,169.551,53.857,160.468
C05122=1007.376,324.961,342.061,169.544,53.862,160.467
C05123=1007.368,324.610,342.106,169.534,53.870,160.467
C05124=1007.359,324.259,342.152,169.522,53.878,160.466
C05125=1007.351,323.908,342.198,169.512,53.885,160.466
C05126=1007.343,323.558,342.243,169.501,53.894,160.466
C05127=1007.337,323.310,342.275,169.494,53.900,160.465
C05128=1007.331,323.062,342.308,169.487,53.905,160.465
C05129=1007.326,322.814,342.340,169.480,53.910,160.465
C05130=1007.321,322.566,342.372,169.472,53.916,160.464
C05131=1007.315,322.318,342.404,169.464,53.922,160.464
C05132=1007.309,322.070,342.436,169.457,53.927,160.464
C05133=1007.303,321.822,342.468,169.450,53.933,160.464
C05134=1007.297,321.575,342.500,169.442,53.938,160.463
C05135=1007.292,321.327,342.533,169.435,53.944,160.463
C05136=1007.287,321.079,342.565,169.427,53.950,160.462
C05137=1007.281,320.831,342.597,169.421,53.955,160.462
C05138=1007.275,320.583,342.628,169.413,53.960,160.462
C05139=1007.270,320.336,342.660,169.405,53.966,160.462
C05140=1007.264,320.088,342.692,169.398,53.972,160.461
C05141=1007.259,319.840,342.724,169.391,53.977,160.461
C05142=1007.253,319.592,342.756,169.384,53.983,160.461
C05143=1007.248,319.344,342.788,169.376,53.989,160.461
C05144=1007.243,319.097,342.820,169.369,53.995,160.460
C05145=1007.237,318.848,342.852,169.362,54.000,160.460
C05146=1007.232,318.600,342.883,169.354,54.005,160.460
C05147=1007.226,318.352,342.915,169.347,54.012,160.460
C05148=1007.221,318.104,342.947,169.341,54.017,160.459
C05149=1007.216,317.857,342.978,169.333,54.023,160.459
C05150=1007.210,317.609,343.010,169.325,54.028,160.459
C05151=1007.204,317.361,343.042,169.318,54.035,160.458
C05152=1007.200,317.112,343.074,169.312,54.040,160.458
C05153=1007.195,316.865,343.105,169.304,54.046,160.458
C05154=1007.189,316.617,343.137,169.296,54.051,160.458
C05155=1007.183,316.369,343.169,169.290,54.057,160.458
C05156=1007.178,316.121,343.200,169.283,54.063,160.457
C05157=1007.173,315.874,343.232,169.275,54.069,160.457
C05158=1007.168,315.626,343.264,169.269,54.074,160.457
C05159=1007.162,315.377,343.295,169.261,54.080,160.457
C05160=1007.157,315.129,343.327,169.254,54.086,160.456
C05161=1007.152,314.882,343.359,169.247,54.092,160.456
C05162=1007.146,314.634,343.390,169.240,54.097,160.456
C05163=1007.141,314.386,343.421,169.233,54.104,160.456
C05164=1007.137,314.138,343.453,169.226,54.109,160.455
C05165=1007.131,313.890,343.484,169.219,54.115,160.455
C05166=1007.126,313.642,343.515,169.211,54.121,160.455
C05167=1007.121,313.395,343.547,169.205,54.127,160.455
C05168=1007.116,313.147,343.578,169.197,54.133,160.455
C05169=1007.110,312.899,343.610,169.190,54.138,160.454
C05170=1007.106,312.651,343.641,169.184,54.144,160.454
C05171=1007.100,312.402,343.673,169.176,54.150,160.454
C05172=1007.095,312.154,343.704,169.169,54.156,160.454
C05173=1007.091,311.907,343.735,169.163,54.162,160.454
C05174=1007.085,311.659,343.766,169.155,54.168,160.453
C05175=1007.081,311.411,343.798,169.149,54.174,160.453
C05176=1007.076,311.163,343.829,169.141,54.179,160.453
C05177=1007.070,310.915,343.860,169.134,54.186,160.453
C05178=1007.065,310.667,343.891,169.128,54.191,160.453
C05179=1007.060,310.419,343.922,169.120,54.197,160.453
C05180=1007.055,310.171,343.954,169.114,54.203,160.453
C05181=1007.050,309.923,343.986,169.107,54.209,160.452
C05182=1007.045,309.675,344.017,169.099,54.215,160.452
C05183=1007.038,309.331,344.060,169.090,54.224,160.452
C05184=1007.032,308.985,344.103,169.080,54.232,160.452
C05185=1007.025,308.640,344.147,169.071,54.240,160.451
C05186=1007.018,308.295,344.189,169.062,54.248,160.451
C05187=1007.014,308.046,344.221,169.055,54.254,160.451
C05188=1007.008,307.799,344.251,169.047,54.261,160.451
C05189=1007.002,307.551,344.281,169.041,54.266,160.451
C05190=1006.997,307.303,344.312,169.034,54.272,160.451
C05191=1006.992,307.055,344.342,169.028,54.278,160.451
C05192=1006.987,306.807,344.372,169.020,54.285,160.450
C05193=1006.982,306.560,344.402,169.013,54.291,160.450
C05194=1006.977,306.311,344.433,169.007,54.297,160.450
C05195=1006.971,306.063,344.463,168.999,54.303,160.450
C05196=1006.966,305.814,344.493,168.993,54.309,160.450
C05197=1006.961,305.567,344.523,168.986,54.315,160.450
C05198=1006.956,305.319,344.554,168.979,54.322,160.450
C05199=1006.950,305.071,344.584,168.973,54.327,160.450
C05200=1006.945,304.822,344.615,168.966,54.334,160.450
C05201=1006.941,304.574,344.645,168.960,54.340,160.450
C05202=1006.935,304.327,344.675,168.953,54.346,160.449
C05203=1006.930,304.027,344.712,168.944,54.353,160.449
C05204=1006.923,303.728,344.747,168.936,54.361,160.449
C05205=1006.918,303.429,344.784,168.928,54.368,160.449
C05206=1006.911,303.131,344.820,168.920,54.376,160.449
C05207=1006.667,303.750,344.379,168.916,54.398,160.453
C05208=1006.676,304.150,344.330,168.926,54.389,160.453
C05209=1006.684,304.549,344.282,168.937,54.379,160.453
C05210=1006.692,304.949,344.234,168.948,54.369,160.454
C05211=1006.701,305.349,344.185,168.960,54.359,160.454
C05212=1006.705,305.597,344.155,168.966,54.353,160.454
C05213=1006.711,305.845,344.124,168.973,54.347,160.454
C05214=1006.715,306.094,344.094,168.979,54.341,160.454
C05215=1006.721,306.342,344.064,168.987,54.335,160.455
C05216=1006.725,306.590,344.034,168.994,54.329,160.455
C05217=1006.731,306.837,344.004,169.000,54.323,160.455
C05218=1006.736,307.086,343.973,169.007,54.317,160.455
C05219=1006.741,307.334,343.942,169.014,54.311,160.455
C05220=1006.746,307.581,343.912,169.021,54.305,160.455
C05221=1006.752,307.829,343.882,169.028,54.298,160.455
C05222=1006.757,308.077,343.851,169.035,54.293,160.456
C05223=1006.762,308.325,343.821,169.042,54.287,160.456
C05224=1006.769,308.673,343.777,169.051,54.279,160.456
C05225=1006.776,309.020,343.734,169.061,54.270,160.456
C05226=1006.782,309.368,343.690,169.071,54.262,160.457
C05227=1006.790,309.715,343.646,169.081,54.254,160.457
C05228=1006.795,309.963,343.615,169.087,54.248,160.457
C05229=1006.798,310.211,343.584,169.094,54.242,160.457
C05230=1006.803,310.459,343.553,169.100,54.236,160.457
C05231=1006.809,310.707,343.522,169.108,54.231,160.458
C05232=1006.814,310.955,343.491,169.114,54.225,160.457
C05233=1006.819,311.203,343.460,169.122,54.219,160.458
C05234=1006.823,311.451,343.428,169.129,54.213,160.458
C05235=1006.828,311.699,343.397,169.136,54.207,160.458
C05236=1006.834,311.947,343.366,169.143,54.201,160.458
C05237=1006.839,312.195,343.335,169.149,54.196,160.459
C05238=1006.844,312.442,343.303,169.157,54.189,160.459
C05239=1006.849,312.691,343.272,169.164,54.184,160.459
C05240=1006.854,312.939,343.240,169.170,54.178,160.459
C05241=1006.859,313.186,343.209,169.178,54.172,160.459
C05242=1006.864,313.435,343.178,169.186,54.166,160.460
C05243=1006.870,313.682,343.146,169.192,54.160,160.460
C05244=1006.875,313.930,343.115,169.199,54.155,160.460
C05245=1006.880,314.178,343.084,169.205,54.149,160.460
C05246=1006.884,314.426,343.052,169.213,54.143,160.461
C05247=1006.890,314.674,343.020,169.221,54.137,160.461
C05248=1006.895,314.922,342.989,169.227,54.131,160.461
C05249=1006.900,315.169,342.958,169.235,54.126,160.461
C05250=1006.905,315.417,342.927,169.242,54.120,160.462
C05251=1006.911,315.665,342.895,169.248,54.114,160.462
C05252=1006.916,315.914,342.863,169.256,54.108,160.462
C05253=1006.921,316.162,342.832,169.264,54.103,160.462
C05254=1006.926,316.409,342.800,169.270,54.098,160.463
C05255=1006.931,316.657,342.769,169.277,54.091,160.463
C05256=1006.937,316.905,342.737,169.285,54.086,160.463
C05257=1006.942,317.153,342.705,169.292,54.080,160.463
C05258=1006.948,317.401,342.673,169.299,54.075,160.464
C05259=1006.953,317.649,342.642,169.306,54.068,160.464
C05260=1006.958,317.896,342.610,169.313,54.063,160.464
C05261=1006.964,318.145,342.578,169.321,54.057,160.464
C05262=1006.969,318.392,342.547,169.328,54.052,160.465
C05263=1006.974,318.640,342.514,169.335,54.046,160.465
C05264=1006.979,318.888,342.484,169.342,54.041,160.465
C05265=1006.985,319.136,342.451,169.350,54.034,160.465
C05266=1006.990,319.384,342.420,169.357,54.029,160.466
C05267=1006.996,319.632,342.388,169.364,54.024,160.466
C05268=1007.002,319.880,342.356,169.372,54.018,160.466
C05269=1007.006,320.127,342.324,169.379,54.012,160.467
C05270=1007.012,320.376,342.292,169.386,54.007,160.467
C05271=1007.018,320.623,342.260,169.393,54.001,160.467
C05272=1007.024,320.871,342.228,169.401,53.996,160.468
C05273=1007.029,321.119,342.197,169.409,53.990,160.468
C05274=1007.034,321.367,342.164,169.415,53.985,160.468
C05275=1007.040,321.615,342.132,169.423,53.979,160.469
C05276=1007.045,321.862,342.101,169.431,53.973,160.469
C05277=1007.051,322.111,342.069,169.438,53.968,160.469
C05278=1007.057,322.358,342.037,169.445,53.963,160.469
C05279=1007.063,322.606,342.005,169.452,53.957,160.470
C05280=1007.068,322.855,341.972,169.460,53.951,160.470
C05281=1007.074,323.102,341.940,169.468,53.946,160.470
C05282=1007.080,323.350,341.908,169.475,53.940,160.471
C05283=1007.085,323.598,341.876,169.482,53.935,160.471
C05284=1007.093,323.951,341.830,169.493,53.927,160.472
C05285=1007.101,324.304,341.785,169.503,53.919,160.472
C05286=1007.110,324.658,341.739,169.514,53.911,160.473
C05287=1007.117,325.011,341.692,169.525,53.904,160.473
C05288=1007.122,325.258,341.659,169.532,53.898,160.473
C05289=1007.128,325.506,341.627,169.540,53.893,160.474
C05290=1007.134,325.754,341.593,169.548,53.888,160.474
C05291=1007.139,326.001,341.561,169.556,53.882,160.475
C05292=1007.145,326.250,341.528,169.562,53.877,160.475
C05293=1007.150,326.498,341.495,169.570,53.871,160.475
C05294=1007.156,326.744,341.463,169.578,53.866,160.476
C05295=1007.161,326.993,341.430,169.586,53.860,160.476
C05296=1007.167,327.241,341.397,169.592,53.855,160.476
C05297=1007.173,327.488,341.364,169.600,53.850,160.477
C05298=1007.178,327.736,341.331,169.608,53.845,160.477
C05299=1007.183,327.984,341.298,169.616,53.839,160.478
C05300=1007.190,328.232,341.266,169.624,53.834,160.478
C05301=1007.195,328.480,341.232,169.631,53.828,160.478
C05302=1007.201,328.727,341.200,169.638,53.824,160.479
C05303=1007.207,328.975,341.166,169.646,53.818,160.479
C05304=1007.212,329.222,341.133,169.654,53.813,160.480
C05305=1007.218,329.470,341.101,169.662,53.808,160.480
C05306=1007.224,329.718,341.067,169.669,53.802,160.480
C05307=1007.229,329.966,341.035,169.678,53.797,160.481
C05308=1007.235,330.214,341.002,169.684,53.792,160.481
C05309=1007.241,330.462,340.969,169.692,53.787,160.482
C05310=1007.246,330.710,340.935,169.700,53.781,160.482
C05311=1007.253,330.957,340.902,169.708,53.776,160.483
C05312=1007.259,331.205,340.868,169.716,53.771,160.483
C05313=1007.264,331.453,340.835,169.724,53.766,160.484
C05314=1007.270,331.701,340.802,169.732,53.761,160.484
C05315=1007.275,331.948,340.768,169.739,53.755,160.484
C05316=1007.281,332.196,340.734,169.747,53.751,160.485
C05317=1007.287,332.443,340.702,169.755,53.746,160.485
C05318=1007.293,332.691,340.668,169.762,53.740,160.486
C05319=1007.299,332.938,340.634,169.770,53.735,160.486
C05320=1007.304,333.186,340.601,169.779,53.730,160.487
C05321=1007.310,333.434,340.568,169.786,53.724,160.487
C05322=1007.316,333.682,340.533,169.794,53.719,160.488
C05323=1007.321,333.929,340.500,169.802,53.715,160.488
C05324=1007.327,334.177,340.466,169.809,53.709,160.489
C05325=1007.333,334.425,340.433,169.817,53.704,160.489
C05326=1007.339,334.672,340.399,169.825,53.699,160.490
C05327=1007.345,334.920,340.366,169.833,53.694,160.490
C05328=1007.351,335.168,340.332,169.841,53.689,160.491
C05329=1007.357,335.415,340.298,169.849,53.684,160.491
C05330=1007.363,335.663,340.264,169.857,53.679,160.492
C05331=1007.369,335.910,340.230,169.865,53.674,160.492
C05332=1007.375,336.159,340.196,169.873,53.669,160.493
C05333=1007.381,336.406,340.162,169.881,53.664,160.493
C05334=1007.386,336.654,340.129,169.889,53.659,160.494
C05335=1007.393,336.901,340.096,169.898,53.654,160.494
C05336=1007.399,337.149,340.061,169.905,53.649,160.495
C05337=1007.405,337.396,340.027,169.913,53.644,160.495
C05338=1007.411,337.643,339.993,169.921,53.639,160.496
C05339=1007.416,337.892,339.959,169.929,53.634,160.496
C05340=1007.422,338.140,339.925,169.938,53.629,160.497
C05341=1007.428,338.387,339.891,169.946,53.624,160.497
C05342=1007.434,338.634,339.857,169.954,53.619,160.498
C05343=1007.440,338.882,339.822,169.962,53.614,160.499
C05344=1007.446,339.098,339.792,169.968,53.610,160.499
C05345=1007.451,339.314,339.762,169.976,53.606,160.500
C05346=1007.456,339.531,339.732,169.983,53.601,160.500
C05347=1007.461,339.747,339.702,169.990,53.598,160.501
C05348=1007.467,339.963,339.672,169.997,53.593,160.501
C05349=1007.472,340.179,339.642,170.005,53.589,160.502
C05350=1007.477,340.395,339.612,170.011,53.585,160.502
C05351=1007.482,340.611,339.582,170.018,53.580,160.503
C05352=1007.489,340.859,339.547,170.026,53.576,160.503
C05353=1007.495,341.106,339.513,170.035,53.571,160.504
C05354=1007.501,341.354,339.479,170.043,53.566,160.504
C05355=1007.507,341.601,339.443,170.051,53.561,160.505
C05356=1007.513,341.849,339.409,170.059,53.556,160.505
C05357=1007.519,342.097,339.375,170.068,53.552,160.506
C05358=1007.526,342.344,339.340,170.077,53.547,160.507
C05359=1007.532,342.591,339.306,170.085,53.542,160.507
C05360=1007.537,342.840,339.271,170.093,53.538,160.508
C05361=1007.543,343.086,339.236,170.101,53.533,160.509
C05362=1007.550,343.334,339.201,170.110,53.528,160.509
C05363=1007.557,343.582,339.166,170.118,53.523,160.510
C05364=1007.562,343.829,339.132,170.126,53.519,160.511
C05365=1007.569,344.077,339.097,170.134,53.514,160.511
C05366=1007.575,344.325,339.062,170.143,53.509,160.512
C05367=1007.581,344.571,339.027,170.151,53.504,160.512
C05368=1007.588,344.819,338.993,170.159,53.500,160.513
C05369=1007.594,345.067,338.957,170.168,53.495,160.514
C05370=1007.600,345.314,338.922,170.176,53.491,160.515
C05371=1007.606,345.562,338.888,170.185,53.486,160.515
C05372=1007.612,345.809,338.852,170.194,53.481,160.516
C05373=1007.619,346.057,338.817,170.202,53.476,160.516
C05374=1007.625,346.304,338.781,170.210,53.472,160.517
C05375=1007.631,346.551,338.747,170.219,53.467,160.518
C05376=1007.637,346.799,338.711,170.227,53.463,160.519
C05377=1007.644,347.046,338.676,170.236,53.459,160.519
C05378=1007.651,347.294,338.641,170.244,53.454,160.520
C05379=1007.657,347.542,338.606,170.252,53.449,160.521
C05380=1007.663,347.789,338.571,170.261,53.444,160.521
C05381=1007.669,348.037,338.535,170.270,53.440,160.522
C05382=1007.676,348.283,338.499,170.279,53.436,160.523
C05383=1007.682,348.530,338.464,170.287,53.431,160.524
C05384=1007.366,346.389,338.411,170.194,53.514,160.524
C05385=1007.359,346.142,338.446,170.186,53.518,160.523
C05386=1007.353,345.894,338.482,170.177,53.523,160.523
C05387=1007.347,345.647,338.516,170.168,53.527,160.522
C05388=1007.341,345.399,338.551,170.160,53.532,160.521
C05389=1007.334,345.152,338.587,170.151,53.537,160.520
C05390=1007.328,344.905,338.621,170.143,53.542,160.520
C05391=1007.322,344.657,338.656,170.135,53.546,160.519
C05392=1007.316,344.410,338.692,170.127,53.551,160.519
C05393=1007.310,344.162,338.726,170.118,53.555,160.518
C05394=1007.303,343.915,338.761,170.110,53.560,160.517
C05395=1007.297,343.667,338.795,170.102,53.564,160.516
C05396=1007.291,343.420,338.831,170.093,53.569,160.516
C05397=1007.285,343.172,338.865,170.085,53.574,160.515
C05398=1007.279,342.925,338.899,170.077,53.578,160.515
C05399=1007.272,342.677,338.934,170.069,53.583,160.514
C05400=1007.266,342.429,338.969,170.059,53.588,160.513
C05401=1007.261,342.182,339.003,170.051,53.593,160.513
C05402=1007.254,341.934,339.038,170.043,53.598,160.512
C05403=1007.248,341.687,339.072,170.034,53.602,160.511
C05404=1007.241,341.439,339.107,170.026,53.607,160.511
C05405=1007.236,341.192,339.142,170.018,53.612,160.510
C05406=1007.230,340.944,339.177,170.010,53.617,160.510
C05407=1007.224,340.697,339.211,170.001,53.621,160.509
C05408=1007.218,340.450,339.245,169.993,53.626,160.508
C05409=1007.208,340.070,339.297,169.982,53.634,160.508
C05410=1007.199,339.691,339.350,169.969,53.641,160.507
C05411=1007.190,339.311,339.403,169.956,53.649,160.506
C05412=1007.180,338.932,339.456,169.944,53.656,160.505
C05413=1007.175,338.684,339.489,169.935,53.661,160.504
C05414=1007.169,338.437,339.523,169.927,53.666,160.504
C05415=1007.163,338.188,339.558,169.919,53.671,160.503
C05416=1007.157,337.941,339.592,169.911,53.676,160.502
C05417=1007.152,337.694,339.626,169.903,53.681,160.502
C05418=1007.145,337.446,339.660,169.896,53.685,160.501
C05419=1007.139,337.198,339.695,169.888,53.690,160.501
C05420=1007.134,336.951,339.728,169.880,53.695,160.500
C05421=1007.128,336.703,339.762,169.871,53.700,160.500
C05422=1007.122,336.456,339.796,169.863,53.705,160.499
C05423=1007.115,336.208,339.829,169.855,53.710,160.499
C05424=1007.109,335.960,339.863,169.847,53.715,160.498
C05425=1007.104,335.713,339.896,169.840,53.720,160.498
C05426=1007.098,335.465,339.931,169.831,53.725,160.497
C05427=1007.092,335.217,339.964,169.823,53.730,160.497
C05428=1007.086,334.969,339.998,169.815,53.735,160.496
C05429=1007.080,334.721,340.032,169.807,53.740,160.496
C05430=1007.074,334.474,340.066,169.799,53.745,160.495
C05431=1007.069,334.226,340.099,169.791,53.750,160.494
C05432=1007.062,333.979,340.132,169.784,53.755,160.494
C05433=1007.057,333.731,340.166,169.776,53.760,160.494
C05434=1007.051,333.484,340.200,169.768,53.765,160.493
C05435=1007.045,333.236,340.233,169.760,53.770,160.493
C05436=1007.040,332.988,340.267,169.752,53.776,160.492
C05437=1007.034,332.740,340.300,169.744,53.781,160.492
C05438=1007.028,332.493,340.334,169.736,53.786,160.491
C05439=1007.023,332.245,340.367,169.728,53.791,160.491
C05440=1007.017,331.997,340.401,169.721,53.796,160.490
C05441=1007.011,331.750,340.434,169.713,53.801,160.490
C05442=1007.005,331.502,340.467,169.705,53.806,160.489
C05443=1006.999,331.255,340.501,169.698,53.812,160.489
C05444=1006.994,331.007,340.534,169.689,53.817,160.488
C05445=1006.988,330.759,340.567,169.682,53.822,160.488
